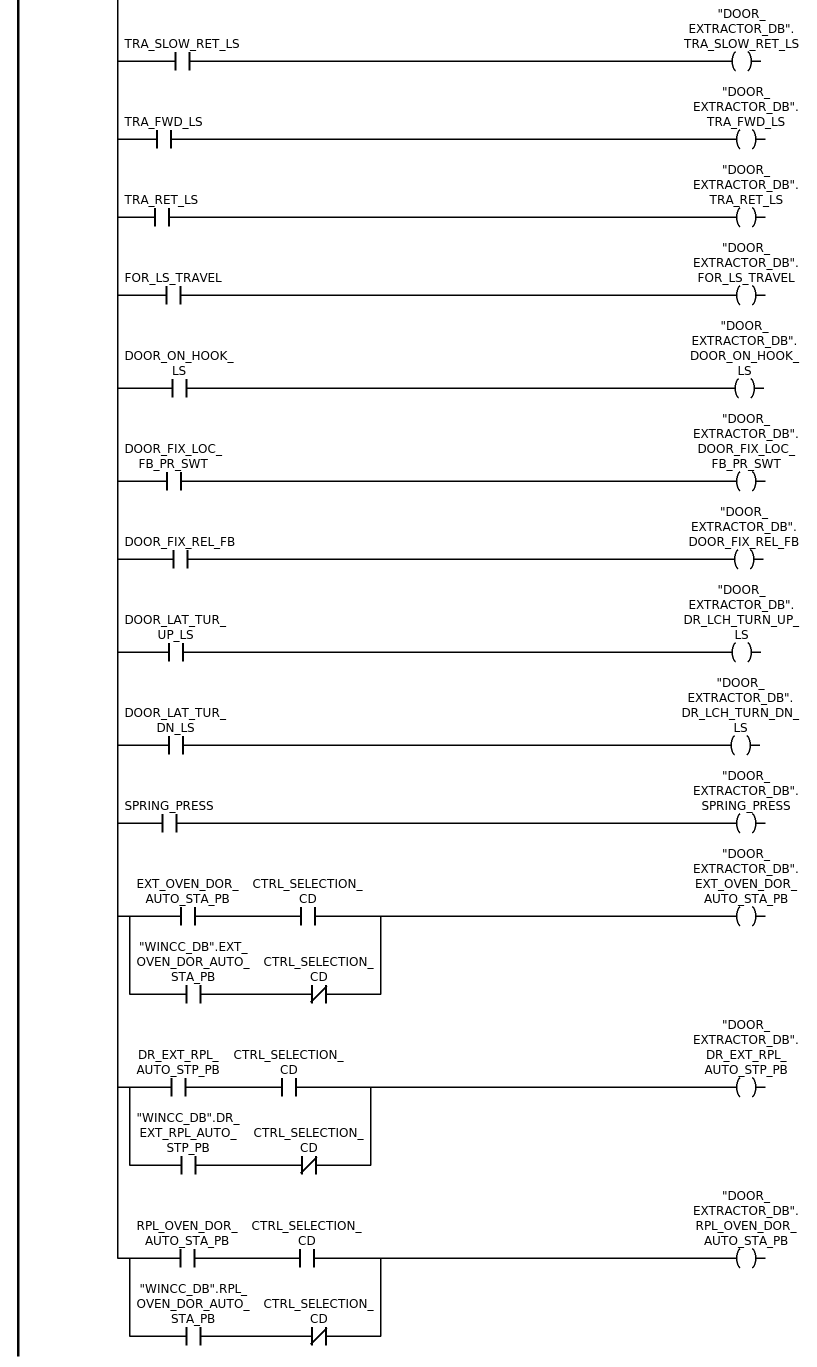
[picture p24: INPUT_MAPPING networks 13-13]
NETWORK
TITLE =
      A     "ALWAYS_ON";
      =     L 0.0;
      A     L 0.0;
      A(;
      O     "DOOR_EXT_LOC_SS";
      O;
      A     "WINCC_DB".REPAIR_MODE_SS;
      AN    "CTRL_SELECTION_CD";
      );
      =     "DOOR_EXTRACTOR_DB".DOOR_EXT_LOC_SS;
      A     L 0.0;
      A(;
      A     "DOOR_EXT_MAN_SS";
      A     "CTRL_SELECTION_CD";
      O;
      A     "WINCC_DB".DE_MAN_SS;
      AN    "DOOR_EXTRACTOR_DB".DOOR_EXT_LOC_SS;
      A     "WINCC_DB".OPER_MODE_SS;
      AN    "CTRL_SELECTION_CD";
      );
      =     "DOOR_EXTRACTOR_DB".DOOR_EXT_MAN_SS;
      A     L 0.0;
      A(;
      A     "DOOR_EXT_AUTO_SS";
      A     "CTRL_SELECTION_CD";
      O;
      A     "WINCC_DB".DE_AUTO_SS;
      AN    "DOOR_EXTRACTOR_DB".DOOR_EXT_LOC_SS;
      A     "WINCC_DB".OPER_MODE_SS;
      AN    "CTRL_SELECTION_CD";
      );
      =     "DOOR_EXTRACTOR_DB".DOOR_EXT_AUTO_SS;
      A     L 0.0;
      A     "WINCC_DB".DE_AUTO_MAN_SS_TAG;
      =     "WINCC_DB".DE_AUTO_SS;
      A     L 0.0;
      AN    "WINCC_DB".DE_AUTO_MAN_SS_TAG;
      =     "WINCC_DB".DE_MAN_SS;
      A     L 0.0;
      A(;
      A     "DOOR_EXT_STP_PB";
      A     "CTRL_SELECTION_CD";
      O;
      A     "WINCC_DB".DE_STP_PB;
      AN    "CTRL_SELECTION_CD";
      );
      =     "DOOR_EXTRACTOR_DB".DOOR_EXT_STP_PB;
      A     L 0.0;
      A(;
      A     "SLEW_FWD_STA_PB";
      A     "CTRL_SELECTION_CD";
      O;
      A     "WINCC_DB".SLEW_FWD_STA_PB;
      AN    "CTRL_SELECTION_CD";
      );
      =     "DOOR_EXTRACTOR_DB".SLEW_FWD_STA_PB;
      A     L 0.0;
      A(;
      A     "SLEW_RET_STA_PB";
      A     "CTRL_SELECTION_CD";
      O;
      A     "WINCC_DB".SLEW_RET_STA_PB;
      AN    "CTRL_SELECTION_CD";
      );
      =     "DOOR_EXTRACTOR_DB".SLEW_RET_STA_PB;
      A     L 0.0;
      A(;
      A     "VER_COMP_FWD_STA";
      A     "CTRL_SELECTION_CD";
      O;
      A     "WINCC_DB".VER_COMP_FWD_STA_PB;
      AN    "CTRL_SELECTION_CD";
      );
      =     "DOOR_EXTRACTOR_DB".VER_COMP_FWD_STA_PB;
      A     L 0.0;
      A(;
      A     "VER_COMP_RET_STA";
      A     "CTRL_SELECTION_CD";
      O;
      A     "WINCC_DB".VER_COMP_RET_STA_PB;
      AN    "CTRL_SELECTION_CD";
      );
      =     "DOOR_EXTRACTOR_DB".VER_COMP_RET_STA_PB;
      A     L 0.0;
      A(;
      A     "TRA_FWD_STA";
      A     "CTRL_SELECTION_CD";
      O;
      A     "WINCC_DB".TRA_FWD_STA_PB;
      AN    "CTRL_SELECTION_CD";
      );
      =     "DOOR_EXTRACTOR_DB".TRA_FWD_STA_PB;
      A     L 0.0;
      A(;
      A     "TRA_RET_STA";
      A     "CTRL_SELECTION_CD";
      O;
      A     "WINCC_DB".TRA_RET_STA_PB;
      AN    "CTRL_SELECTION_CD";
      );
      =     "DOOR_EXTRACTOR_DB".TRA_RET_STA_PB;
      A     L 0.0;
      A(;
      A     "MAN_STK_UP_STA_PB";
      A     "CTRL_SELECTION_CD";
      O;
      A     "WINCC_DB".MAIN_STK_UP_STA_PB;
      AN    "CTRL_SELECTION_CD";
      );
      =     "DOOR_EXTRACTOR_DB".MAIN_STK_UP_STA_PB;
      A     L 0.0;
      A(;
      A     "MAN_STK_UP_DN_PB";
      A     "CTRL_SELECTION_CD";
      O;
      A     "WINCC_DB".MAIN_STK_UP_DN_PB;
      AN    "CTRL_SELECTION_CD";
      );
      =     "DOOR_EXTRACTOR_DB".MAIN_STK_UP_DN_PB;
      A     L 0.0;
      A(;
      A     "FNL_STK_UP_STA_PB";
      A     "CTRL_SELECTION_CD";
      O;
      A     "WINCC_DB".FIN_STK_UP_STA_PB;
      AN    "CTRL_SELECTION_CD";
      );
      =     "DOOR_EXTRACTOR_DB".FIN_STK_UP_STA_PB;
      A     L 0.0;
      A(;
      A     "FNL_STK_UP_DN_PB";
      A     "CTRL_SELECTION_CD";
      O;
      A     "WINCC_DB".FIN_STK_UP_DN_PB;
      AN    "CTRL_SELECTION_CD";
      );
      =     "DOOR_EXTRACTOR_DB".FIN_STK_UP_DN_PB;
      A     L 0.0;
      A(;
      A     "PRE_STK_UP_STA_PB";
      A     "CTRL_SELECTION_CD";
      O;
      A     "WINCC_DB".PRE_STK_UP_STA_PB;
      AN    "CTRL_SELECTION_CD";
      );
      =     "DOOR_EXTRACTOR_DB".PRE_STK_UP_STA_PB;
      A     L 0.0;
      A(;
      A     "PRE_STK_UP_DN_PB";
      A     "CTRL_SELECTION_CD";
      O;
      A     "WINCC_DB".PRE_STK_UP_DN_PB;
      AN    "CTRL_SELECTION_CD";
      );
      =     "DOOR_EXTRACTOR_DB".PRE_STK_UP_DN_PB;
      A     L 0.0;
      A(;
      A     "DOOR_SPRG_PRS_STA_PB";
      A     "CTRL_SELECTION_CD";
      O;
      A     "WINCC_DB".DR_SPNG_LK_STA_PB;
      AN    "CTRL_SELECTION_CD";
      );
      =     "DOOR_EXTRACTOR_DB".DR_SPNG_LK_STA_PB;
      A     L 0.0;
      A(;
      A     "DOOR_SPRG_RLES_STA_PB";
      A     "CTRL_SELECTION_CD";
      O;
      A     "WINCC_DB".DR_SPNG_UNLK_STA_PB;
      AN    "CTRL_SELECTION_CD";
      );
      =     "DOOR_EXTRACTOR_DB".DR_SPNG_UNLK_STA_PB;
      A     L 0.0;
      A(;
      A     "DOOR_LCH_TURN_LOCK";
      A     "CTRL_SELECTION_CD";
      O;
      A     "WINCC_DB".DR_LCH_TURN_UP_PB;
      AN    "CTRL_SELECTION_CD";
      );
      =     "DOOR_EXTRACTOR_DB".DR_LCH_TURN_UP_PB;
      A     L 0.0;
      A(;
      A     "DOOR_LCH_TURN_UNLOC";
      A     "CTRL_SELECTION_CD";
      O;
      A     "WINCC_DB".DR_LCH_TURN_DN_PB;
      AN    "CTRL_SELECTION_CD";
      );
      =     "DOOR_EXTRACTOR_DB".DR_LCH_TURN_DN_PB;
      A     L 0.0;
      A     "EMERGENCY_PB_LCS_73";
      =     "DOOR_EXTRACTOR_DB".EMERGENCY_PB_LCS_73;
      A     L 0.0;
      A     "SLEW_FWD_STA_LCS";
      =     "DOOR_EXTRACTOR_DB".SLEW_FWD_STA_PB_LCS;
      A     L 0.0;
      A     "SLEW_RET_STA_LCS";
      =     "DOOR_EXTRACTOR_DB".SLEW_RET_STA_PB_LCS;
      A     L 0.0;
      A     "VER_COMP_FWD_STA_LCS";
      =     "DOOR_EXTRACTOR_DB".VER_COMP_FWD_STA_PB_LCS;
      A     L 0.0;
      A     "VER_COMP_RET_STA_LCS";
      =     "DOOR_EXTRACTOR_DB".VER_COMP_RET_STA_PB_LCS;
      A     L 0.0;
      A     "TRA_FWD_STA_LCS";
      =     "DOOR_EXTRACTOR_DB".TRA_FWD_STA_PB_LCS;
      A     L 0.0;
      A     "TRA_BACK_STA_LCS";
      =     "DOOR_EXTRACTOR_DB".TRA_RET_STA_PB_LCS;
      A     L 0.0;
      A     "MAIN_STK_UP_STA_LCS";
      =     "DOOR_EXTRACTOR_DB".MAIN_STK_UP_STA_PB_LCS;
      A     L 0.0;
      A     "MAIN_STK_DN_STA_LCS";
      =     "DOOR_EXTRACTOR_DB".MAIN_STK_DN_STA_PB_LCS;
      A     L 0.0;
      A     "FNL_STK_UP_STA_LCS";
      =     "DOOR_EXTRACTOR_DB".FIN_STK_UP_STA_PB_LCS;
      A     L 0.0;
      A     "FNL_STK_DN_STA_LCS";
      =     "DOOR_EXTRACTOR_DB".FIN_STK_DN_STA_PB_LCS;
      A     L 0.0;
      A     "PRE_STK_UP_STA_LCS";
      =     "DOOR_EXTRACTOR_DB".PRE_STK_UP_STA_PB_LCS;
      A     L 0.0;
      A     "PRE_STK_DN_STA_LCS";
      =     "DOOR_EXTRACTOR_DB".PRE_STK_DN_STA_PB_LCS;
      A     L 0.0;
      A     "DOOR_SPRG_PRS_LK_STA_LCS";
      =     "DOOR_EXTRACTOR_DB".DR_SPNG_LK_STA_PB_LCS;
      A     L 0.0;
      A     "DOOR_SPRG_RLES_UNLSTA_LC";
      =     "DOOR_EXTRACTOR_DB".DR_SPNG_UNLK_STA_PB_LCS;
      A     L 0.0;
      A     "LAMP_TEST_PB_LCS_73";
      =     "DOOR_EXTRACTOR_DB".LAMP_TEST_PB_LCS_73;
      A     L 0.0;
      A     "DOOR_LAT_LOCK_PB_LCS";
      =     "DOOR_EXTRACTOR_DB".DR_LCH_TURN_UP_PB_LCS;
      A     L 0.0;
      A     "DOOR_LAT_UNLOCK_PB_LCS1";
      =     "DOOR_EXTRACTOR_DB".DR_LCH_TURN_DN_PB_LCS;
      A     L 0.0;
      A     "DOOR_LAT_HOME_PB_LCS";
      =     "DOOR_EXTRACTOR_DB".DR_LCH_TURN_HOME_PB_LCS;
      A     L 0.0;
      A     "SLEW_SLOW_FWD_LS";
      =     "DOOR_EXTRACTOR_DB".SLEW_SLOW_FWD_LS;
      A     L 0.0;
      A     "SLEW_SLOW_RET_LS";
      =     "DOOR_EXTRACTOR_DB".SLEW_SLOW_RET_LS;
      A     L 0.0;
      A     "SLEW_NOR_FWD_LS";
      =     "DOOR_EXTRACTOR_DB".SLEW_NOR_FWD_LS;
      A     L 0.0;
      A     "SLEW_NOR_RET_LS";
      =     "DOOR_EXTRACTOR_DB".SLEW_NOR_RET_LS;
      A     L 0.0;
      A     "TRA_SLOW_FWD_LS";
      =     "DOOR_EXTRACTOR_DB".TRA_SLOW_FWD_LS;
      A     L 0.0;
      A     "TRA_SLOW_RET_LS";
      =     "DOOR_EXTRACTOR_DB".TRA_SLOW_RET_LS;
      A     L 0.0;
      A     "TRA_FWD_LS";
      =     "DOOR_EXTRACTOR_DB".TRA_FWD_LS;
      A     L 0.0;
      A     "TRA_RET_LS";
      =     "DOOR_EXTRACTOR_DB".TRA_RET_LS;
      A     L 0.0;
      A     "FOR_LS_TRAVEL";
      =     "DOOR_EXTRACTOR_DB".FOR_LS_TRAVEL;
      A     L 0.0;
      A     "DOOR_ON_HOOK_LS";
      =     "DOOR_EXTRACTOR_DB".DOOR_ON_HOOK_LS;
      A     L 0.0;
      A     "DOOR_FIX_LOC_FB_PR_SWT";
      =     "DOOR_EXTRACTOR_DB".DOOR_FIX_LOC_FB_PR_SWT;
      A     L 0.0;
      A     "DOOR_FIX_REL_FB";
      =     "DOOR_EXTRACTOR_DB".DOOR_FIX_REL_FB;
      A     L 0.0;
      A     "DOOR_LAT_TUR_UP_LS";
      =     "DOOR_EXTRACTOR_DB".DR_LCH_TURN_UP_LS;
      A     L 0.0;
      A     "DOOR_LAT_TUR_DN_LS";
      =     "DOOR_EXTRACTOR_DB".DR_LCH_TURN_DN_LS;
      A     L 0.0;
      A     "SPRING_PRESS";
      =     "DOOR_EXTRACTOR_DB".SPRING_PRESS;
      A     L 0.0;
      A(;
      A     "EXT_OVEN_DOR_AUTO_STA_PB";
      A     "CTRL_SELECTION_CD";
      O;
      A     "WINCC_DB".EXT_OVEN_DOR_AUTO_STA_PB;
      AN    "CTRL_SELECTION_CD";
      );
      =     "DOOR_EXTRACTOR_DB".EXT_OVEN_DOR_AUTO_STA_PB;
      A     L 0.0;
      A(;
      A     "DR_EXT_RPL_AUTO_STP_PB";
      A     "CTRL_SELECTION_CD";
      O;
      A     "WINCC_DB".DR_EXT_RPL_AUTO_STP_PB;
      AN    "CTRL_SELECTION_CD";
      );
      =     "DOOR_EXTRACTOR_DB".DR_EXT_RPL_AUTO_STP_PB;
      A     L 0.0;
      A(;
      A     "RPL_OVEN_DOR_AUTO_STA_PB";
      A     "CTRL_SELECTION_CD";
      O;
      A     "WINCC_DB".RPL_OVEN_DOR_AUTO_STA_PB;
      AN    "CTRL_SELECTION_CD";
      );
      =     "DOOR_EXTRACTOR_DB".RPL_OVEN_DOR_AUTO_STA_PB;
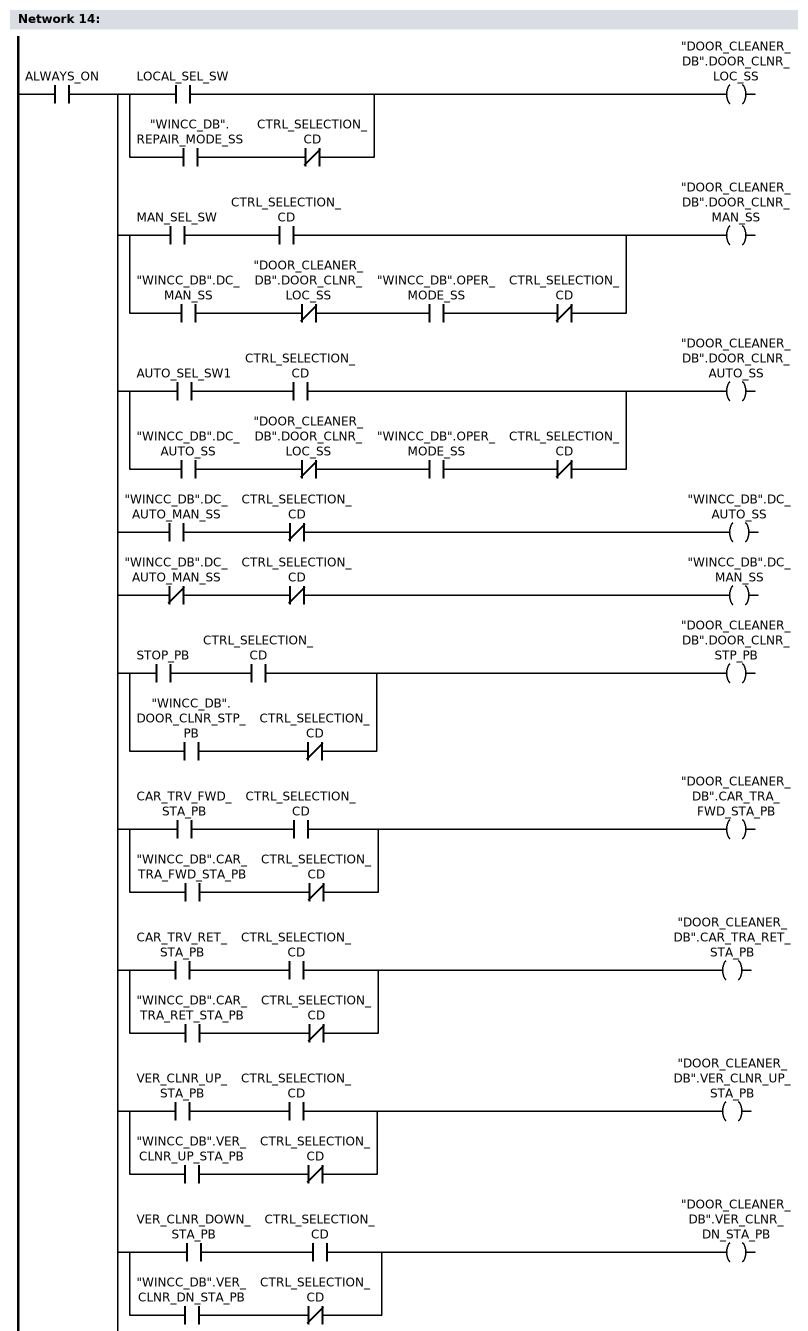
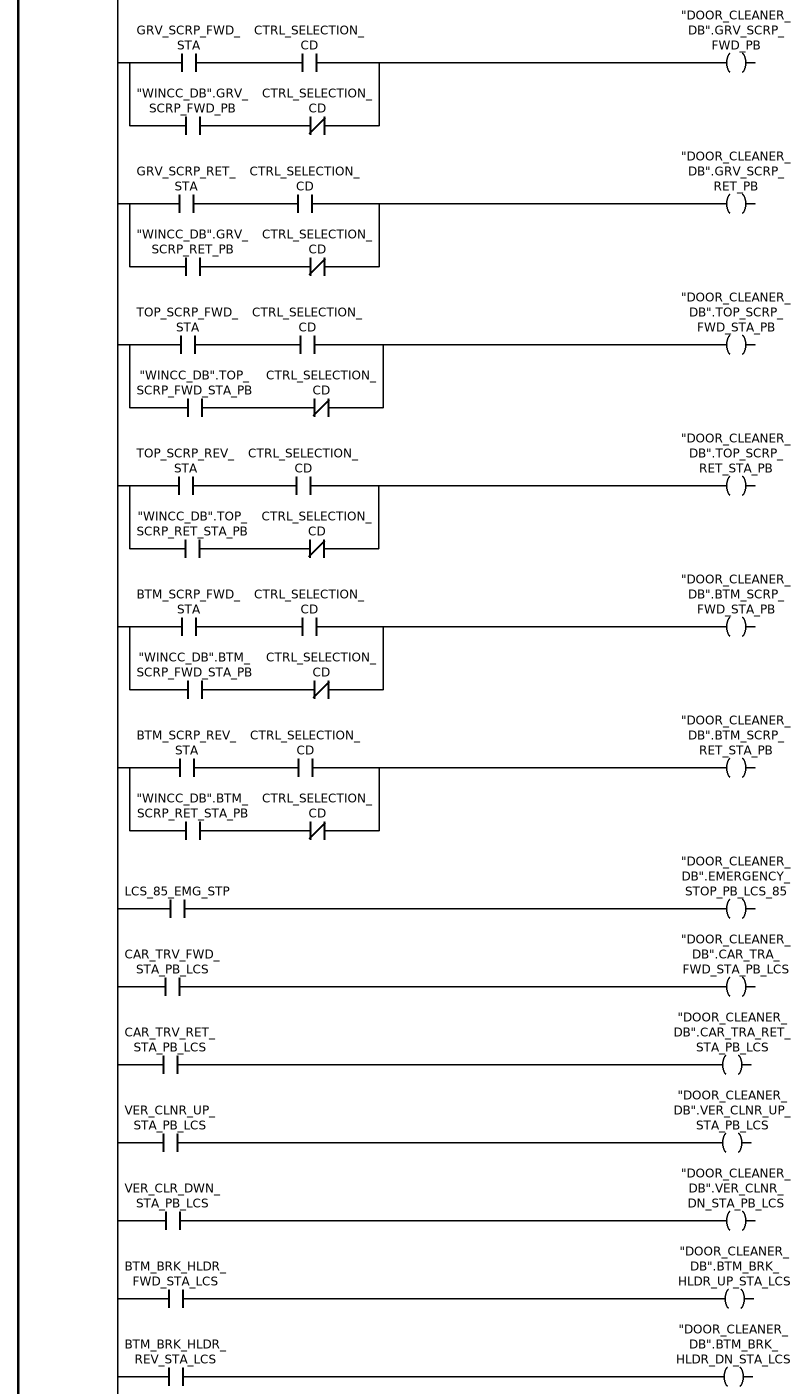
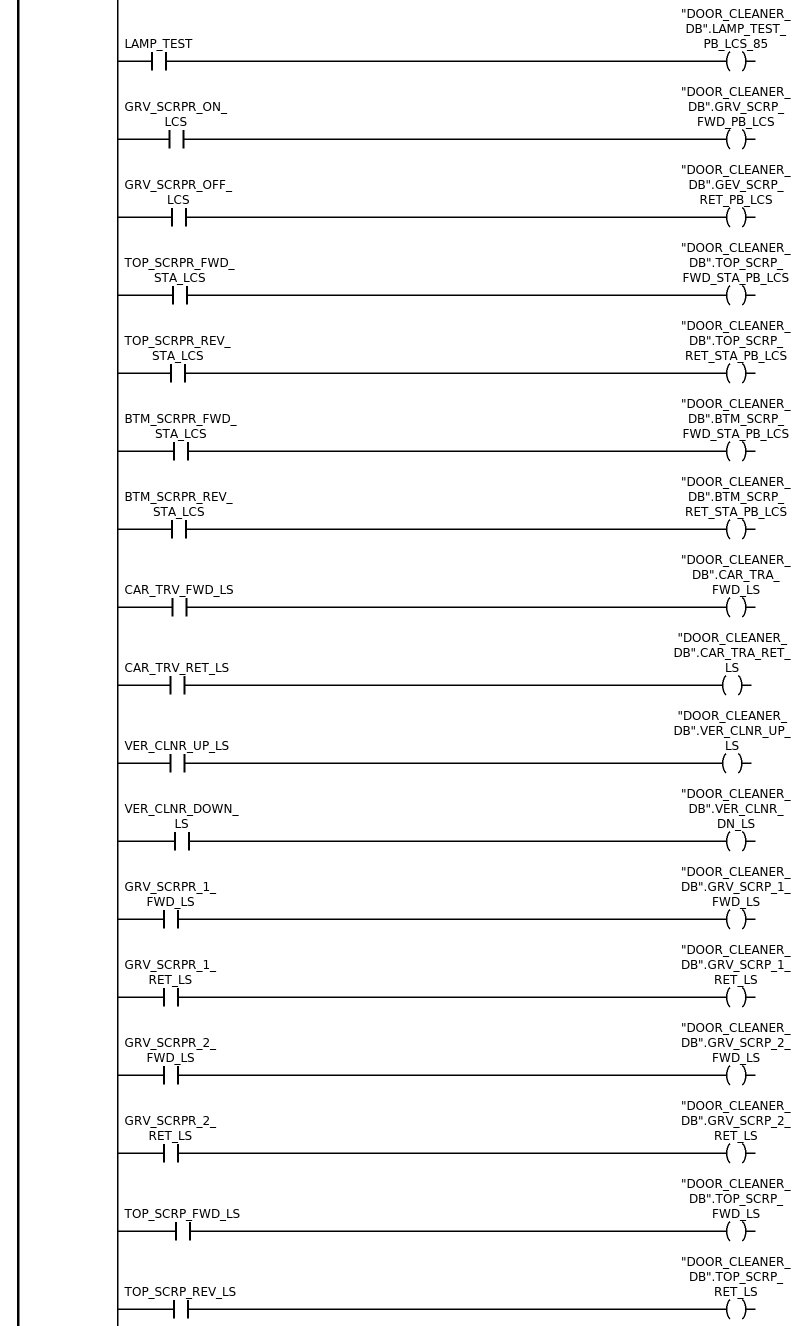
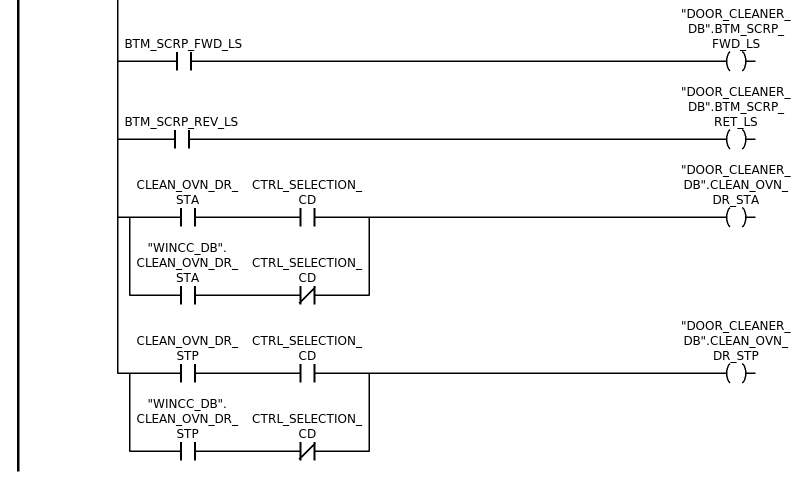
NETWORK
TITLE =
      A     "ALWAYS_ON";
      =     L 0.0;
      A     L 0.0;
      A(;
      O     "LOCAL_SEL_SW";
      O;
      A     "WINCC_DB".REPAIR_MODE_SS;
      AN    "CTRL_SELECTION_CD";
      );
      =     "DOOR_CLEANER_DB".DOOR_CLNR_LOC_SS;
      A     L 0.0;
      A(;
      A     "MAN_SEL_SW";
      A     "CTRL_SELECTION_CD";
      O;
      A     "WINCC_DB".DC_MAN_SS;
      AN    "DOOR_CLEANER_DB".DOOR_CLNR_LOC_SS;
      A     "WINCC_DB".OPER_MODE_SS;
      AN    "CTRL_SELECTION_CD";
      );
      =     "DOOR_CLEANER_DB".DOOR_CLNR_MAN_SS;
      A     L 0.0;
      A(;
      A     "AUTO_SEL_SW1";
      A     "CTRL_SELECTION_CD";
      O;
      A     "WINCC_DB".DC_AUTO_SS;
      AN    "DOOR_CLEANER_DB".DOOR_CLNR_LOC_SS;
      A     "WINCC_DB".OPER_MODE_SS;
      AN    "CTRL_SELECTION_CD";
      );
      =     "DOOR_CLEANER_DB".DOOR_CLNR_AUTO_SS;
      A     L 0.0;
      A     "WINCC_DB".DC_AUTO_MAN_SS;
      AN    "CTRL_SELECTION_CD";
      =     "WINCC_DB".DC_AUTO_SS;
      A     L 0.0;
      AN    "WINCC_DB".DC_AUTO_MAN_SS;
      AN    "CTRL_SELECTION_CD";
      =     "WINCC_DB".DC_MAN_SS;
      A     L 0.0;
      A(;
      A     "STOP_PB";
      A     "CTRL_SELECTION_CD";
      O;
      A     "WINCC_DB".DOOR_CLNR_STP_PB;
      AN    "CTRL_SELECTION_CD";
      );
      =     "DOOR_CLEANER_DB".DOOR_CLNR_STP_PB;
      A     L 0.0;
      A(;
      A     "CAR_TRV_FWD_STA_PB";
      A     "CTRL_SELECTION_CD";
      O;
      A     "WINCC_DB".CAR_TRA_FWD_STA_PB;
      AN    "CTRL_SELECTION_CD";
      );
      =     "DOOR_CLEANER_DB".CAR_TRA_FWD_STA_PB;
      A     L 0.0;
      A(;
      A     "CAR_TRV_RET_STA_PB";
      A     "CTRL_SELECTION_CD";
      O;
      A     "WINCC_DB".CAR_TRA_RET_STA_PB;
      AN    "CTRL_SELECTION_CD";
      );
      =     "DOOR_CLEANER_DB".CAR_TRA_RET_STA_PB;
      A     L 0.0;
      A(;
      A     "VER_CLNR_UP_STA_PB";
      A     "CTRL_SELECTION_CD";
      O;
      A     "WINCC_DB".VER_CLNR_UP_STA_PB;
      AN    "CTRL_SELECTION_CD";
      );
      =     "DOOR_CLEANER_DB".VER_CLNR_UP_STA_PB;
      A     L 0.0;
      A(;
      A     "VER_CLNR_DOWN_STA_PB";
      A     "CTRL_SELECTION_CD";
      O;
      A     "WINCC_DB".VER_CLNR_DN_STA_PB;
      AN    "CTRL_SELECTION_CD";
      );
      =     "DOOR_CLEANER_DB".VER_CLNR_DN_STA_PB;
      A     L 0.0;
      A(;
      A     "GRV_SCRP_FWD_STA";
      A     "CTRL_SELECTION_CD";
      O;
      A     "WINCC_DB".GRV_SCRP_FWD_PB;
      AN    "CTRL_SELECTION_CD";
      );
      =     "DOOR_CLEANER_DB".GRV_SCRP_FWD_PB;
      A     L 0.0;
      A(;
      A     "GRV_SCRP_RET_STA";
      A     "CTRL_SELECTION_CD";
      O;
      A     "WINCC_DB".GRV_SCRP_RET_PB;
      AN    "CTRL_SELECTION_CD";
      );
      =     "DOOR_CLEANER_DB".GRV_SCRP_RET_PB;
      A     L 0.0;
      A(;
      A     "TOP_SCRP_FWD_STA";
      A     "CTRL_SELECTION_CD";
      O;
      A     "WINCC_DB".TOP_SCRP_FWD_STA_PB;
      AN    "CTRL_SELECTION_CD";
      );
      =     "DOOR_CLEANER_DB".TOP_SCRP_FWD_STA_PB;
      A     L 0.0;
      A(;
      A     "TOP_SCRP_REV_STA";
      A     "CTRL_SELECTION_CD";
      O;
      A     "WINCC_DB".TOP_SCRP_RET_STA_PB;
      AN    "CTRL_SELECTION_CD";
      );
      =     "DOOR_CLEANER_DB".TOP_SCRP_RET_STA_PB;
      A     L 0.0;
      A(;
      A     "BTM_SCRP_FWD_STA";
      A     "CTRL_SELECTION_CD";
      O;
      A     "WINCC_DB".BTM_SCRP_FWD_STA_PB;
      AN    "CTRL_SELECTION_CD";
      );
      =     "DOOR_CLEANER_DB".BTM_SCRP_FWD_STA_PB;
      A     L 0.0;
      A(;
      A     "BTM_SCRP_REV_STA";
      A     "CTRL_SELECTION_CD";
      O;
      A     "WINCC_DB".BTM_SCRP_RET_STA_PB;
      AN    "CTRL_SELECTION_CD";
      );
      =     "DOOR_CLEANER_DB".BTM_SCRP_RET_STA_PB;
      A     L 0.0;
      A     "LCS_85_EMG_STP";
      =     "DOOR_CLEANER_DB".EMERGENCY_STOP_PB_LCS_85;
      A     L 0.0;
      A     "CAR_TRV_FWD_STA_PB_LCS";
      =     "DOOR_CLEANER_DB".CAR_TRA_FWD_STA_PB_LCS;
      A     L 0.0;
      A     "CAR_TRV_RET_STA_PB_LCS";
      =     "DOOR_CLEANER_DB".CAR_TRA_RET_STA_PB_LCS;
      A     L 0.0;
      A     "VER_CLNR_UP_STA_PB_LCS";
      =     "DOOR_CLEANER_DB".VER_CLNR_UP_STA_PB_LCS;
      A     L 0.0;
      A     "VER_CLR_DWN_STA_PB_LCS";
      =     "DOOR_CLEANER_DB".VER_CLNR_DN_STA_PB_LCS;
      A     L 0.0;
      A     "BTM_BRK_HLDR_FWD_STA_LCS";
      =     "DOOR_CLEANER_DB".BTM_BRK_HLDR_UP_STA_LCS;
      A     L 0.0;
      A     "BTM_BRK_HLDR_REV_STA_LCS";
      =     "DOOR_CLEANER_DB".BTM_BRK_HLDR_DN_STA_LCS;
      A     L 0.0;
      A     "LAMP_TEST";
      =     "DOOR_CLEANER_DB".LAMP_TEST_PB_LCS_85;
      A     L 0.0;
      A     "GRV_SCRPR_ON_LCS";
      =     "DOOR_CLEANER_DB".GRV_SCRP_FWD_PB_LCS;
      A     L 0.0;
      A     "GRV_SCRPR_OFF_LCS";
      =     "DOOR_CLEANER_DB".GEV_SCRP_RET_PB_LCS;
      A     L 0.0;
      A     "TOP_SCRPR_FWD_STA_LCS";
      =     "DOOR_CLEANER_DB".TOP_SCRP_FWD_STA_PB_LCS;
      A     L 0.0;
      A     "TOP_SCRPR_REV_STA_LCS";
      =     "DOOR_CLEANER_DB".TOP_SCRP_RET_STA_PB_LCS;
      A     L 0.0;
      A     "BTM_SCRPR_FWD_STA_LCS";
      =     "DOOR_CLEANER_DB".BTM_SCRP_FWD_STA_PB_LCS;
      A     L 0.0;
      A     "BTM_SCRPR_REV_STA_LCS";
      =     "DOOR_CLEANER_DB".BTM_SCRP_RET_STA_PB_LCS;
      A     L 0.0;
      A     "CAR_TRV_FWD_LS";
      =     "DOOR_CLEANER_DB".CAR_TRA_FWD_LS;
      A     L 0.0;
      A     "CAR_TRV_RET_LS";
      =     "DOOR_CLEANER_DB".CAR_TRA_RET_LS;
      A     L 0.0;
      A     "VER_CLNR_UP_LS";
      =     "DOOR_CLEANER_DB".VER_CLNR_UP_LS;
      A     L 0.0;
      A     "VER_CLNR_DOWN_LS";
      =     "DOOR_CLEANER_DB".VER_CLNR_DN_LS;
      A     L 0.0;
      A     "GRV_SCRPR_1_FWD_LS";
      =     "DOOR_CLEANER_DB".GRV_SCRP_1_FWD_LS;
      A     L 0.0;
      A     "GRV_SCRPR_1_RET_LS";
      =     "DOOR_CLEANER_DB".GRV_SCRP_1_RET_LS;
      A     L 0.0;
      A     "GRV_SCRPR_2_FWD_LS";
      =     "DOOR_CLEANER_DB".GRV_SCRP_2_FWD_LS;
      A     L 0.0;
      A     "GRV_SCRPR_2_RET_LS";
      =     "DOOR_CLEANER_DB".GRV_SCRP_2_RET_LS;
      A     L 0.0;
      A     "TOP_SCRP_FWD_LS";
      =     "DOOR_CLEANER_DB".TOP_SCRP_FWD_LS;
      A     L 0.0;
      A     "TOP_SCRP_REV_LS";
      =     "DOOR_CLEANER_DB".TOP_SCRP_RET_LS;
      A     L 0.0;
      A     "BTM_SCRP_FWD_LS";
      =     "DOOR_CLEANER_DB".BTM_SCRP_FWD_LS;
      A     L 0.0;
      A     "BTM_SCRP_REV_LS";
      =     "DOOR_CLEANER_DB".BTM_SCRP_RET_LS;
      A     L 0.0;
      A(;
      A     "CLEAN_OVN_DR_STA";
      A     "CTRL_SELECTION_CD";
      O;
      A     "WINCC_DB".CLEAN_OVN_DR_STA;
      AN    "CTRL_SELECTION_CD";
      );
      =     "DOOR_CLEANER_DB".CLEAN_OVN_DR_STA;
      A     L 0.0;
      A(;
      A     "CLEAN_OVN_DR_STP";
      A     "CTRL_SELECTION_CD";
      O;
      A     "WINCC_DB".CLEAN_OVN_DR_STP;
      AN    "CTRL_SELECTION_CD";
      );
      =     "DOOR_CLEANER_DB".CLEAN_OVN_DR_STP;
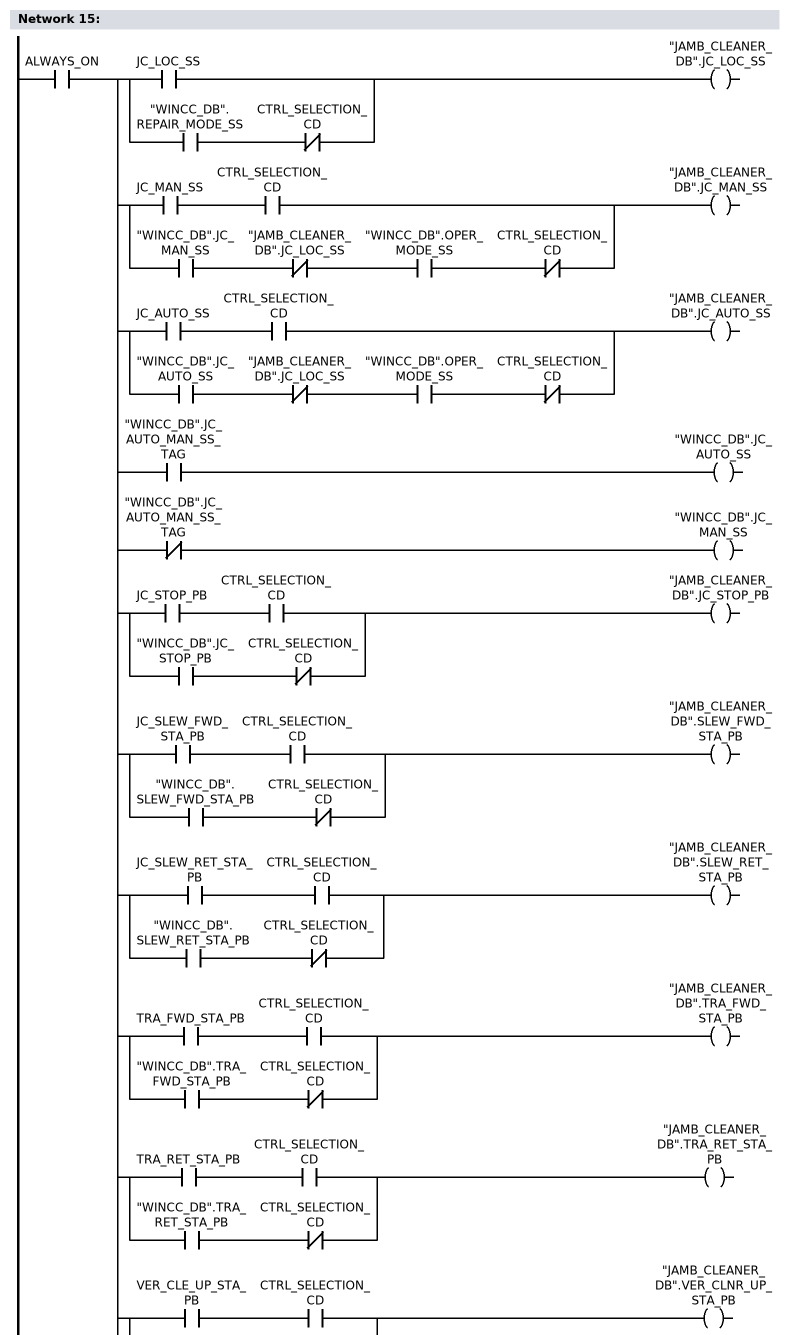
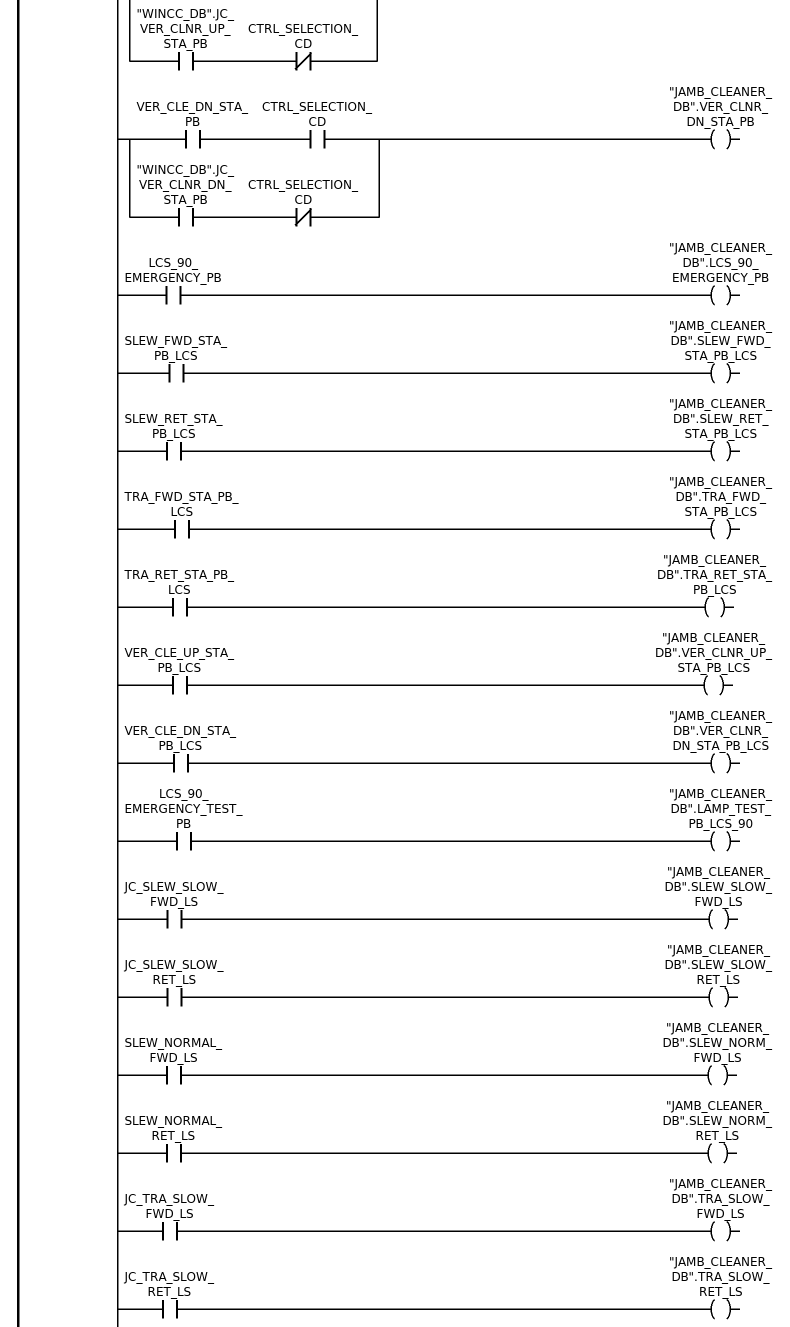
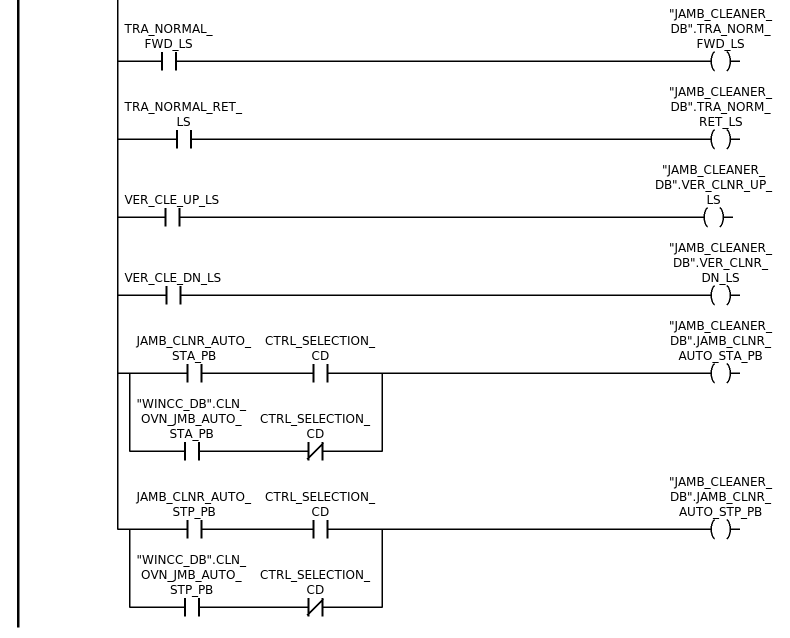
NETWORK
TITLE =
      A     "ALWAYS_ON";
      =     L 0.0;
      A     L 0.0;
      A(;
      O     "JC_LOC_SS";
      O;
      A     "WINCC_DB".REPAIR_MODE_SS;
      AN    "CTRL_SELECTION_CD";
      );
      =     "JAMB_CLEANER_DB".JC_LOC_SS;
      A     L 0.0;
      A(;
      A     "JC_MAN_SS";
      A     "CTRL_SELECTION_CD";
      O;
      A     "WINCC_DB".JC_MAN_SS;
      AN    "JAMB_CLEANER_DB".JC_LOC_SS;
      A     "WINCC_DB".OPER_MODE_SS;
      AN    "CTRL_SELECTION_CD";
      );
      =     "JAMB_CLEANER_DB".JC_MAN_SS;
      A     L 0.0;
      A(;
      A     "JC_AUTO_SS";
      A     "CTRL_SELECTION_CD";
      O;
      A     "WINCC_DB".JC_AUTO_SS;
      AN    "JAMB_CLEANER_DB".JC_LOC_SS;
      A     "WINCC_DB".OPER_MODE_SS;
      AN    "CTRL_SELECTION_CD";
      );
      =     "JAMB_CLEANER_DB".JC_AUTO_SS;
      A     L 0.0;
      A     "WINCC_DB".JC_AUTO_MAN_SS_TAG;
      =     "WINCC_DB".JC_AUTO_SS;
      A     L 0.0;
      AN    "WINCC_DB".JC_AUTO_MAN_SS_TAG;
      =     "WINCC_DB".JC_MAN_SS;
      A     L 0.0;
      A(;
      A     "JC_STOP_PB";
      A     "CTRL_SELECTION_CD";
      O;
      A     "WINCC_DB".JC_STOP_PB;
      AN    "CTRL_SELECTION_CD";
      );
      =     "JAMB_CLEANER_DB".JC_STOP_PB;
      A     L 0.0;
      A(;
      A     "JC_SLEW_FWD_STA_PB";
      A     "CTRL_SELECTION_CD";
      O;
      A     "WINCC_DB".SLEW_FWD_STA_PB;
      AN    "CTRL_SELECTION_CD";
      );
      =     "JAMB_CLEANER_DB".SLEW_FWD_STA_PB;
      A     L 0.0;
      A(;
      A     "JC_SLEW_RET_STA_PB";
      A     "CTRL_SELECTION_CD";
      O;
      A     "WINCC_DB".SLEW_RET_STA_PB;
      AN    "CTRL_SELECTION_CD";
      );
      =     "JAMB_CLEANER_DB".SLEW_RET_STA_PB;
      A     L 0.0;
      A(;
      A     "TRA_FWD_STA_PB";
      A     "CTRL_SELECTION_CD";
      O;
      A     "WINCC_DB".TRA_FWD_STA_PB;
      AN    "CTRL_SELECTION_CD";
      );
      =     "JAMB_CLEANER_DB".TRA_FWD_STA_PB;
      A     L 0.0;
      A(;
      A     "TRA_RET_STA_PB";
      A     "CTRL_SELECTION_CD";
      O;
      A     "WINCC_DB".TRA_RET_STA_PB;
      AN    "CTRL_SELECTION_CD";
      );
      =     "JAMB_CLEANER_DB".TRA_RET_STA_PB;
      A     L 0.0;
      A(;
      A     "VER_CLE_UP_STA_PB";
      A     "CTRL_SELECTION_CD";
      O;
      A     "WINCC_DB".JC_VER_CLNR_UP_STA_PB;
      AN    "CTRL_SELECTION_CD";
      );
      =     "JAMB_CLEANER_DB".VER_CLNR_UP_STA_PB;
      A     L 0.0;
      A(;
      A     "VER_CLE_DN_STA_PB";
      A     "CTRL_SELECTION_CD";
      O;
      A     "WINCC_DB".JC_VER_CLNR_DN_STA_PB;
      AN    "CTRL_SELECTION_CD";
      );
      =     "JAMB_CLEANER_DB".VER_CLNR_DN_STA_PB;
      A     L 0.0;
      A     "LCS_90_EMERGENCY_PB";
      =     "JAMB_CLEANER_DB".LCS_90_EMERGENCY_PB;
      A     L 0.0;
      A     "SLEW_FWD_STA_PB_LCS";
      =     "JAMB_CLEANER_DB".SLEW_FWD_STA_PB_LCS;
      A     L 0.0;
      A     "SLEW_RET_STA_PB_LCS";
      =     "JAMB_CLEANER_DB".SLEW_RET_STA_PB_LCS;
      A     L 0.0;
      A     "TRA_FWD_STA_PB_LCS";
      =     "JAMB_CLEANER_DB".TRA_FWD_STA_PB_LCS;
      A     L 0.0;
      A     "TRA_RET_STA_PB_LCS";
      =     "JAMB_CLEANER_DB".TRA_RET_STA_PB_LCS;
      A     L 0.0;
      A     "VER_CLE_UP_STA_PB_LCS";
      =     "JAMB_CLEANER_DB".VER_CLNR_UP_STA_PB_LCS;
      A     L 0.0;
      A     "VER_CLE_DN_STA_PB_LCS";
      =     "JAMB_CLEANER_DB".VER_CLNR_DN_STA_PB_LCS;
      A     L 0.0;
      A     "LCS_90_EMERGENCY_TEST_PB";
      =     "JAMB_CLEANER_DB".LAMP_TEST_PB_LCS_90;
      A     L 0.0;
      A     "JC_SLEW_SLOW_FWD_LS";
      =     "JAMB_CLEANER_DB".SLEW_SLOW_FWD_LS;
      A     L 0.0;
      A     "JC_SLEW_SLOW_RET_LS";
      =     "JAMB_CLEANER_DB".SLEW_SLOW_RET_LS;
      A     L 0.0;
      A     "SLEW_NORMAL_FWD_LS";
      =     "JAMB_CLEANER_DB".SLEW_NORM_FWD_LS;
      A     L 0.0;
      A     "SLEW_NORMAL_RET_LS";
      =     "JAMB_CLEANER_DB".SLEW_NORM_RET_LS;
      A     L 0.0;
      A     "JC_TRA_SLOW_FWD_LS";
      =     "JAMB_CLEANER_DB".TRA_SLOW_FWD_LS;
      A     L 0.0;
      A     "JC_TRA_SLOW_RET_LS";
      =     "JAMB_CLEANER_DB".TRA_SLOW_RET_LS;
      A     L 0.0;
      A     "TRA_NORMAL_FWD_LS";
      =     "JAMB_CLEANER_DB".TRA_NORM_FWD_LS;
      A     L 0.0;
      A     "TRA_NORMAL_RET_LS";
      =     "JAMB_CLEANER_DB".TRA_NORM_RET_LS;
      A     L 0.0;
      A     "VER_CLE_UP_LS";
      =     "JAMB_CLEANER_DB".VER_CLNR_UP_LS;
      A     L 0.0;
      A     "VER_CLE_DN_LS";
      =     "JAMB_CLEANER_DB".VER_CLNR_DN_LS;
      A     L 0.0;
      A(;
      A     "JAMB_CLNR_AUTO_STA_PB";
      A     "CTRL_SELECTION_CD";
      O;
      A     "WINCC_DB".CLN_OVN_JMB_AUTO_STA_PB;
      AN    "CTRL_SELECTION_CD";
      );
      =     "JAMB_CLEANER_DB".JAMB_CLNR_AUTO_STA_PB;
      A     L 0.0;
      A(;
      A     "JAMB_CLNR_AUTO_STP_PB";
      A     "CTRL_SELECTION_CD";
      O;
      A     "WINCC_DB".CLN_OVN_JMB_AUTO_STP_PB;
      AN    "CTRL_SELECTION_CD";
      );
      =     "JAMB_CLEANER_DB".JAMB_CLNR_AUTO_STP_PB;
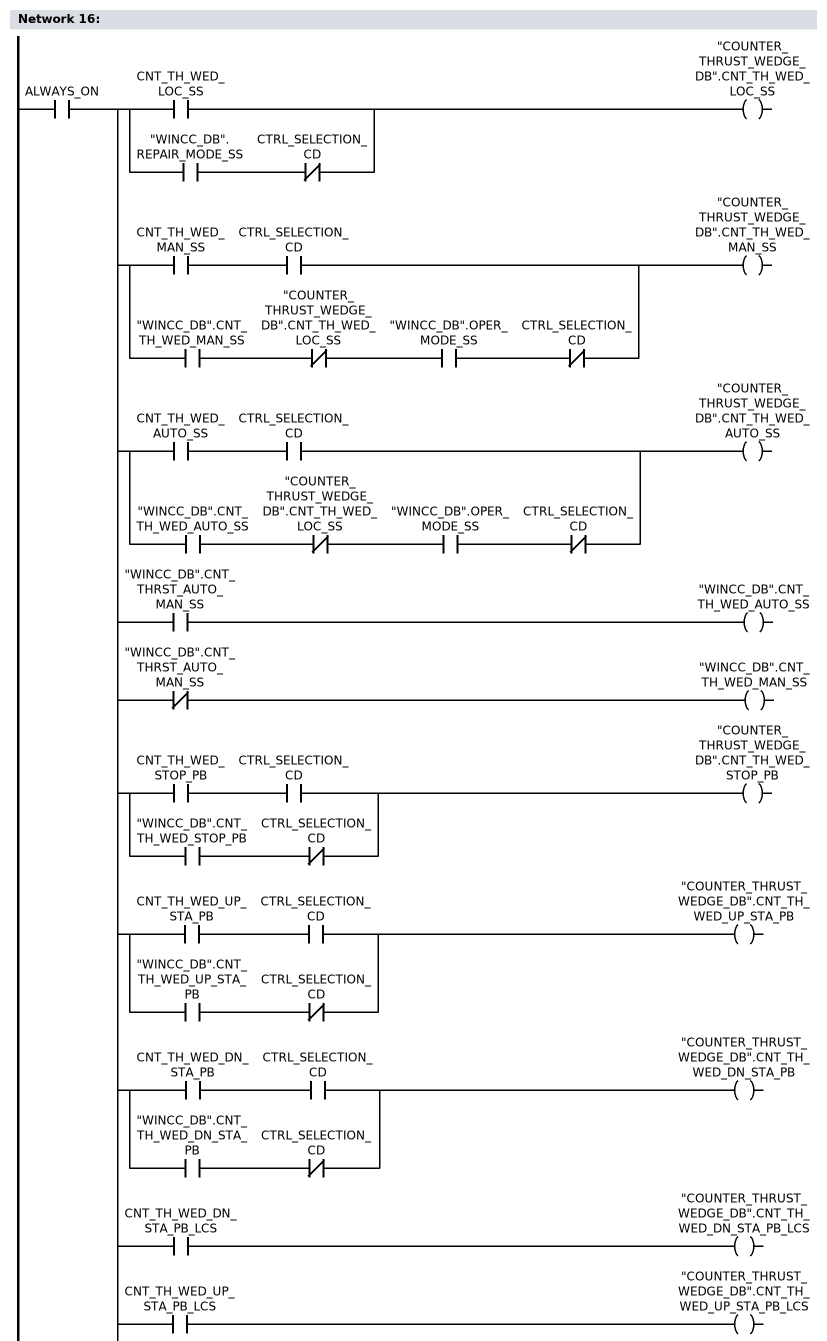
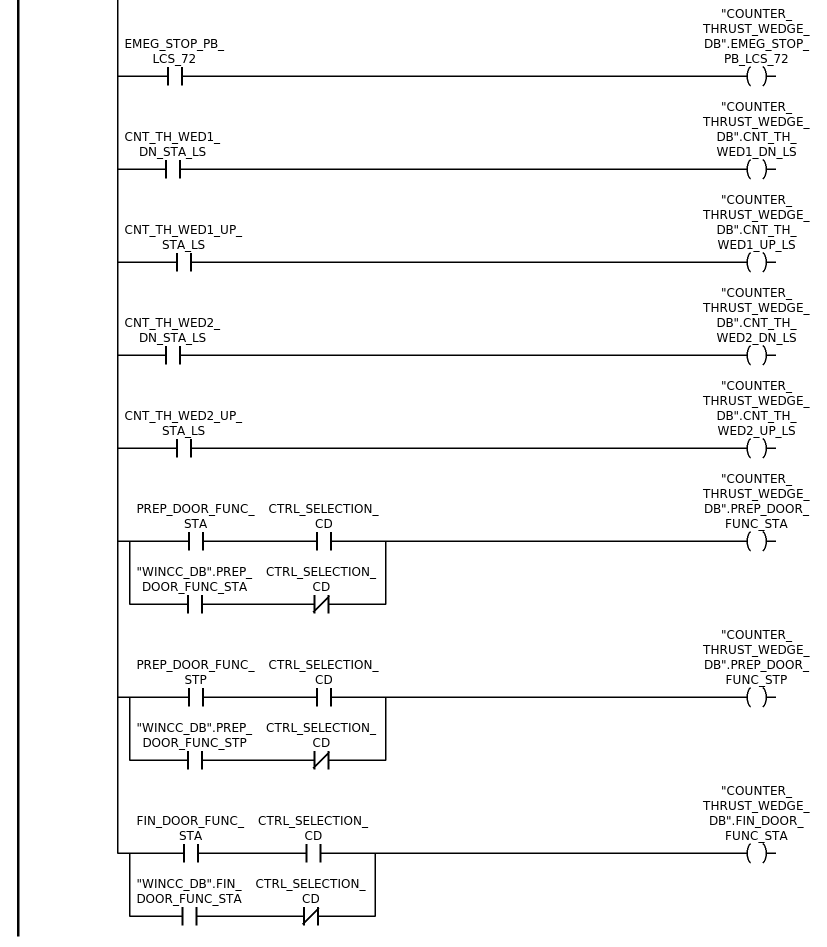
NETWORK
TITLE =
      A     "ALWAYS_ON";
      =     L 0.0;
      A     L 0.0;
      A(;
      O     "CNT_TH_WED_LOC_SS";
      O;
      A     "WINCC_DB".REPAIR_MODE_SS;
      AN    "CTRL_SELECTION_CD";
      );
      =     "COUNTER_THRUST_WEDGE_DB".CNT_TH_WED_LOC_SS;
      A     L 0.0;
      A(;
      A     "CNT_TH_WED_MAN_SS";
      A     "CTRL_SELECTION_CD";
      O;
      A     "WINCC_DB".CNT_TH_WED_MAN_SS;
      AN    "COUNTER_THRUST_WEDGE_DB".CNT_TH_WED_LOC_SS;
      A     "WINCC_DB".OPER_MODE_SS;
      AN    "CTRL_SELECTION_CD";
      );
      =     "COUNTER_THRUST_WEDGE_DB".CNT_TH_WED_MAN_SS;
      A     L 0.0;
      A(;
      A     "CNT_TH_WED_AUTO_SS";
      A     "CTRL_SELECTION_CD";
      O;
      A     "WINCC_DB".CNT_TH_WED_AUTO_SS;
      AN    "COUNTER_THRUST_WEDGE_DB".CNT_TH_WED_LOC_SS;
      A     "WINCC_DB".OPER_MODE_SS;
      AN    "CTRL_SELECTION_CD";
      );
      =     "COUNTER_THRUST_WEDGE_DB".CNT_TH_WED_AUTO_SS;
      A     L 0.0;
      A     "WINCC_DB".CNT_THRST_AUTO_MAN_SS;
      =     "WINCC_DB".CNT_TH_WED_AUTO_SS;
      A     L 0.0;
      AN    "WINCC_DB".CNT_THRST_AUTO_MAN_SS;
      =     "WINCC_DB".CNT_TH_WED_MAN_SS;
      A     L 0.0;
      A(;
      A     "CNT_TH_WED_STOP_PB";
      A     "CTRL_SELECTION_CD";
      O;
      A     "WINCC_DB".CNT_TH_WED_STOP_PB;
      AN    "CTRL_SELECTION_CD";
      );
      =     "COUNTER_THRUST_WEDGE_DB".CNT_TH_WED_STOP_PB;
      A     L 0.0;
      A(;
      A     "CNT_TH_WED_UP_STA_PB";
      A     "CTRL_SELECTION_CD";
      O;
      A     "WINCC_DB".CNT_TH_WED_UP_STA_PB;
      AN    "CTRL_SELECTION_CD";
      );
      =     "COUNTER_THRUST_WEDGE_DB".CNT_TH_WED_UP_STA_PB;
      A     L 0.0;
      A(;
      A     "CNT_TH_WED_DN_STA_PB";
      A     "CTRL_SELECTION_CD";
      O;
      A     "WINCC_DB".CNT_TH_WED_DN_STA_PB;
      AN    "CTRL_SELECTION_CD";
      );
      =     "COUNTER_THRUST_WEDGE_DB".CNT_TH_WED_DN_STA_PB;
      A     L 0.0;
      A     "CNT_TH_WED_DN_STA_PB_LCS";
      =     "COUNTER_THRUST_WEDGE_DB".CNT_TH_WED_DN_STA_PB_LCS;
      A     L 0.0;
      A     "CNT_TH_WED_UP_STA_PB_LCS";
      =     "COUNTER_THRUST_WEDGE_DB".CNT_TH_WED_UP_STA_PB_LCS;
      A     L 0.0;
      A     "EMEG_STOP_PB_LCS_72";
      =     "COUNTER_THRUST_WEDGE_DB".EMEG_STOP_PB_LCS_72;
      A     L 0.0;
      A     "CNT_TH_WED1_DN_STA_LS";
      =     "COUNTER_THRUST_WEDGE_DB".CNT_TH_WED1_DN_LS;
      A     L 0.0;
      A     "CNT_TH_WED1_UP_STA_LS";
      =     "COUNTER_THRUST_WEDGE_DB".CNT_TH_WED1_UP_LS;
      A     L 0.0;
      A     "CNT_TH_WED2_DN_STA_LS";
      =     "COUNTER_THRUST_WEDGE_DB".CNT_TH_WED2_DN_LS;
      A     L 0.0;
      A     "CNT_TH_WED2_UP_STA_LS";
      =     "COUNTER_THRUST_WEDGE_DB".CNT_TH_WED2_UP_LS;
      A     L 0.0;
      A(;
      A     "PREP_DOOR_FUNC_STA";
      A     "CTRL_SELECTION_CD";
      O;
      A     "WINCC_DB".PREP_DOOR_FUNC_STA;
      AN    "CTRL_SELECTION_CD";
      );
      =     "COUNTER_THRUST_WEDGE_DB".PREP_DOOR_FUNC_STA;
      A     L 0.0;
      A(;
      A     "PREP_DOOR_FUNC_STP";
      A     "CTRL_SELECTION_CD";
      O;
      A     "WINCC_DB".PREP_DOOR_FUNC_STP;
      AN    "CTRL_SELECTION_CD";
      );
      =     "COUNTER_THRUST_WEDGE_DB".PREP_DOOR_FUNC_STP;
      A     L 0.0;
      A(;
      A     "FIN_DOOR_FUNC_STA";
      A     "CTRL_SELECTION_CD";
      O;
      A     "WINCC_DB".FIN_DOOR_FUNC_STA;
      AN    "CTRL_SELECTION_CD";
      );
      =     "COUNTER_THRUST_WEDGE_DB".FIN_DOOR_FUNC_STA;
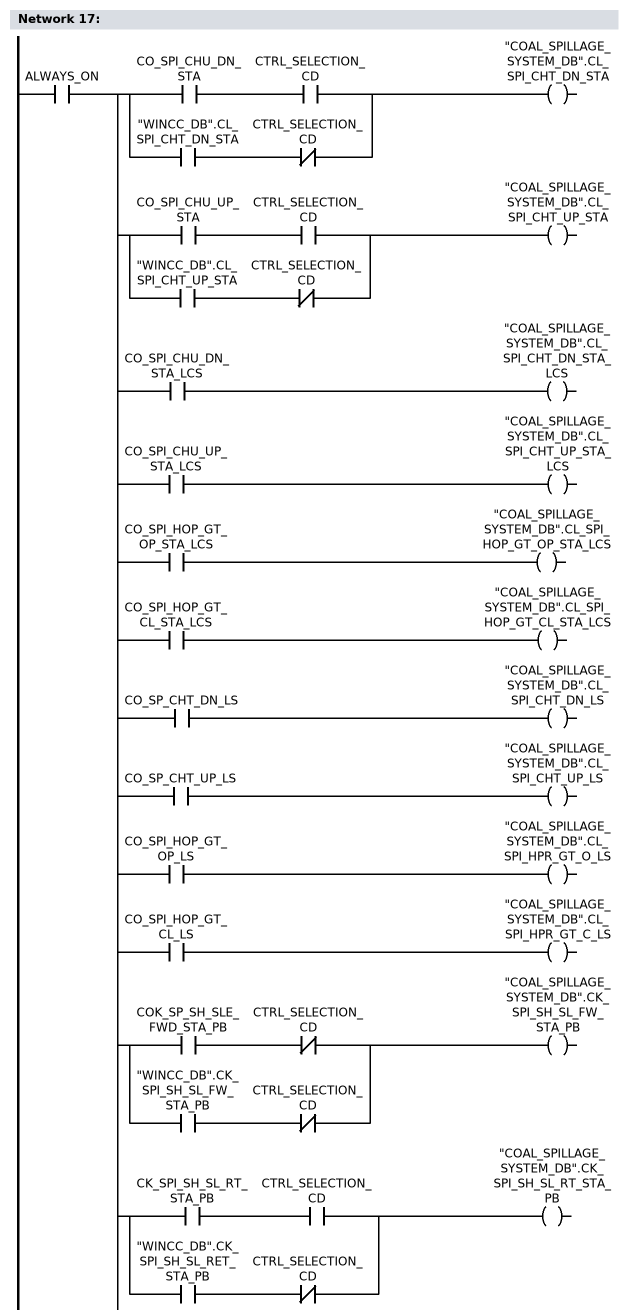
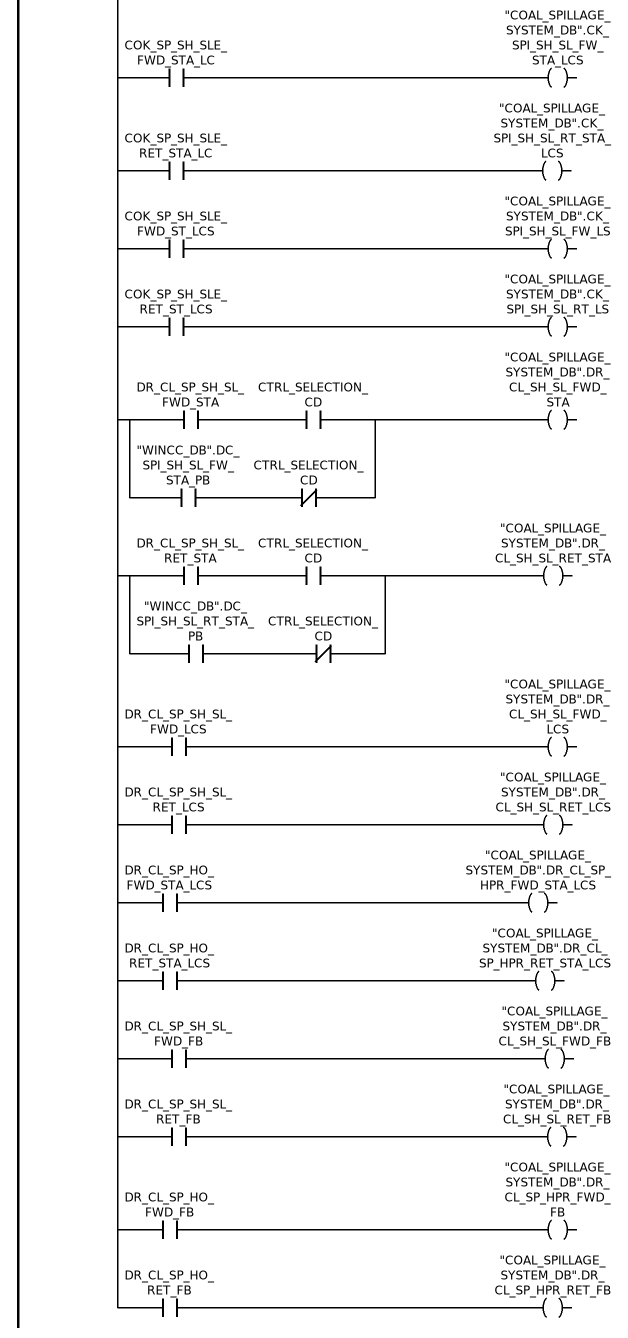
NETWORK
TITLE =
      A     "ALWAYS_ON";
      =     L 0.0;
      A     L 0.0;
      A(;
      A     "CO_SPI_CHU_DN_STA";
      A     "CTRL_SELECTION_CD";
      O;
      A     "WINCC_DB".CL_SPI_CHT_DN_STA;
      AN    "CTRL_SELECTION_CD";
      );
      =     "COAL_SPILLAGE_SYSTEM_DB".CL_SPI_CHT_DN_STA;
      A     L 0.0;
      A(;
      A     "CO_SPI_CHU_UP_STA";
      A     "CTRL_SELECTION_CD";
      O;
      A     "WINCC_DB".CL_SPI_CHT_UP_STA;
      AN    "CTRL_SELECTION_CD";
      );
      =     "COAL_SPILLAGE_SYSTEM_DB".CL_SPI_CHT_UP_STA;
      A     L 0.0;
      A     "CO_SPI_CHU_DN_STA_LCS";
      =     "COAL_SPILLAGE_SYSTEM_DB".CL_SPI_CHT_DN_STA_LCS;
      A     L 0.0;
      A     "CO_SPI_CHU_UP_STA_LCS";
      =     "COAL_SPILLAGE_SYSTEM_DB".CL_SPI_CHT_UP_STA_LCS;
      A     L 0.0;
      A     "CO_SPI_HOP_GT_OP_STA_LCS";
      =     "COAL_SPILLAGE_SYSTEM_DB".CL_SPI_HOP_GT_OP_STA_LCS;
      A     L 0.0;
      A     "CO_SPI_HOP_GT_CL_STA_LCS";
      =     "COAL_SPILLAGE_SYSTEM_DB".CL_SPI_HOP_GT_CL_STA_LCS;
      A     L 0.0;
      A     "CO_SP_CHT_DN_LS";
      =     "COAL_SPILLAGE_SYSTEM_DB".CL_SPI_CHT_DN_LS;
      A     L 0.0;
      A     "CO_SP_CHT_UP_LS";
      =     "COAL_SPILLAGE_SYSTEM_DB".CL_SPI_CHT_UP_LS;
      A     L 0.0;
      A     "CO_SPI_HOP_GT_OP_LS";
      =     "COAL_SPILLAGE_SYSTEM_DB".CL_SPI_HPR_GT_O_LS;
      A     L 0.0;
      A     "CO_SPI_HOP_GT_CL_LS";
      =     "COAL_SPILLAGE_SYSTEM_DB".CL_SPI_HPR_GT_C_LS;
      A     L 0.0;
      A(;
      A     "COK_SP_SH_SLE_FWD_STA_PB";
      AN    "CTRL_SELECTION_CD";
      O;
      A     "WINCC_DB".CK_SPI_SH_SL_FW_STA_PB;
      AN    "CTRL_SELECTION_CD";
      );
      =     "COAL_SPILLAGE_SYSTEM_DB".CK_SPI_SH_SL_FW_STA_PB;
      A     L 0.0;
      A(;
      A     "CK_SPI_SH_SL_RT_STA_PB";
      A     "CTRL_SELECTION_CD";
      O;
      A     "WINCC_DB".CK_SPI_SH_SL_RET_STA_PB;
      AN    "CTRL_SELECTION_CD";
      );
      =     "COAL_SPILLAGE_SYSTEM_DB".CK_SPI_SH_SL_RT_STA_PB;
      A     L 0.0;
      A     "COK_SP_SH_SLE_FWD_STA_LC";
      =     "COAL_SPILLAGE_SYSTEM_DB".CK_SPI_SH_SL_FW_STA_LCS;
      A     L 0.0;
      A     "COK_SP_SH_SLE_RET_STA_LC";
      =     "COAL_SPILLAGE_SYSTEM_DB".CK_SPI_SH_SL_RT_STA_LCS;
      A     L 0.0;
      A     "COK_SP_SH_SLE_FWD_ST_LCS";
      =     "COAL_SPILLAGE_SYSTEM_DB".CK_SPI_SH_SL_FW_LS;
      A     L 0.0;
      A     "COK_SP_SH_SLE_RET_ST_LCS";
      =     "COAL_SPILLAGE_SYSTEM_DB".CK_SPI_SH_SL_RT_LS;
      A     L 0.0;
      A(;
      A     "DR_CL_SP_SH_SL_FWD_STA";
      A     "CTRL_SELECTION_CD";
      O;
      A     "WINCC_DB".DC_SPI_SH_SL_FW_STA_PB;
      AN    "CTRL_SELECTION_CD";
      );
      =     "COAL_SPILLAGE_SYSTEM_DB".DR_CL_SH_SL_FWD_STA;
      A     L 0.0;
      A(;
      A     "DR_CL_SP_SH_SL_RET_STA";
      A     "CTRL_SELECTION_CD";
      O;
      A     "WINCC_DB".DC_SPI_SH_SL_RT_STA_PB;
      AN    "CTRL_SELECTION_CD";
      );
      =     "COAL_SPILLAGE_SYSTEM_DB".DR_CL_SH_SL_RET_STA;
      A     L 0.0;
      A     "DR_CL_SP_SH_SL_FWD_LCS";
      =     "COAL_SPILLAGE_SYSTEM_DB".DR_CL_SH_SL_FWD_LCS;
      A     L 0.0;
      A     "DR_CL_SP_SH_SL_RET_LCS";
      =     "COAL_SPILLAGE_SYSTEM_DB".DR_CL_SH_SL_RET_LCS;
      A     L 0.0;
      A     "DR_CL_SP_HO_FWD_STA_LCS";
      =     "COAL_SPILLAGE_SYSTEM_DB".DR_CL_SP_HPR_FWD_STA_LCS;
      A     L 0.0;
      A     "DR_CL_SP_HO_RET_STA_LCS";
      =     "COAL_SPILLAGE_SYSTEM_DB".DR_CL_SP_HPR_RET_STA_LCS;
      A     L 0.0;
      A     "DR_CL_SP_SH_SL_FWD_FB";
      =     "COAL_SPILLAGE_SYSTEM_DB".DR_CL_SH_SL_FWD_FB;
      A     L 0.0;
      A     "DR_CL_SP_SH_SL_RET_FB";
      =     "COAL_SPILLAGE_SYSTEM_DB".DR_CL_SH_SL_RET_FB;
      A     L 0.0;
      A     "DR_CL_SP_HO_FWD_FB";
      =     "COAL_SPILLAGE_SYSTEM_DB".DR_CL_SP_HPR_FWD_FB;
      A     L 0.0;
      A     "DR_CL_SP_HO_RET_FB";
      =     "COAL_SPILLAGE_SYSTEM_DB".DR_CL_SP_HPR_RET_FB;
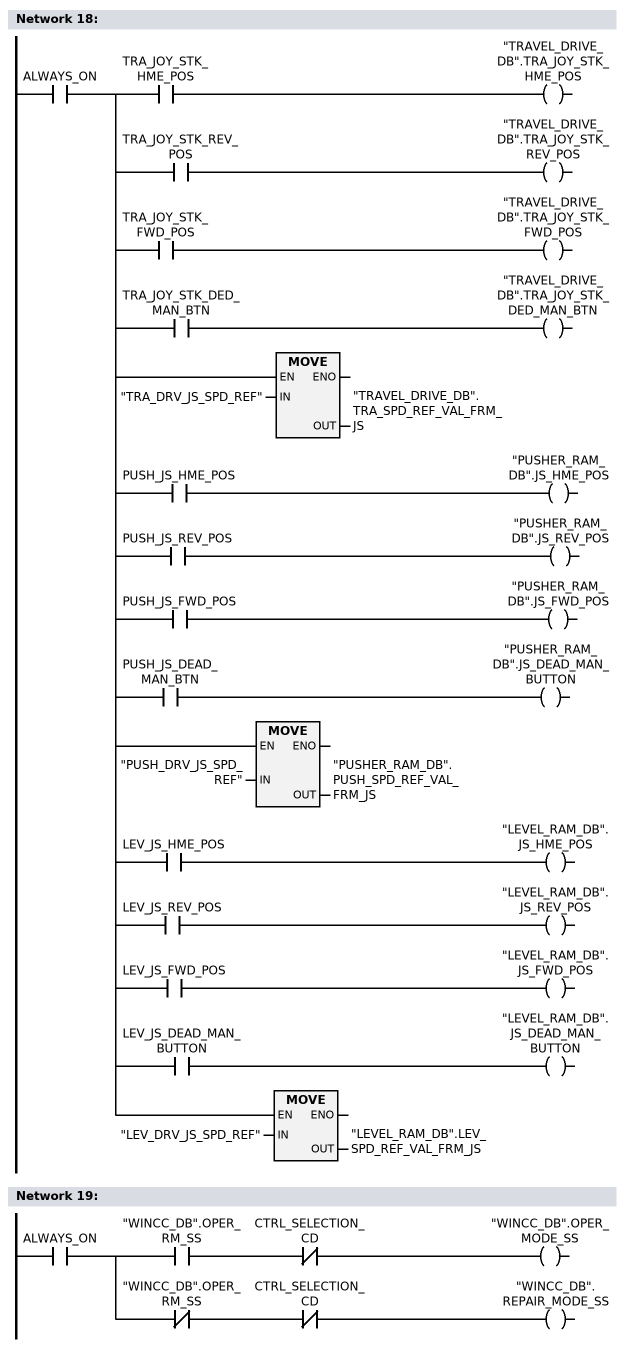
NETWORK
TITLE =
      A     "ALWAYS_ON";
      =     L 0.0;
      A     L 0.0;
      A     "TRA_JOY_STK_HME_POS";
      =     "TRAVEL_DRIVE_DB".TRA_JOY_STK_HME_POS;
      A     L 0.0;
      A     "TRA_JOY_STK_REV_POS";
      =     "TRAVEL_DRIVE_DB".TRA_JOY_STK_REV_POS;
      A     L 0.0;
      A     "TRA_JOY_STK_FWD_POS";
      =     "TRAVEL_DRIVE_DB".TRA_JOY_STK_FWD_POS;
      A     L 0.0;
      A     "TRA_JOY_STK_DED_MAN_BTN";
      =     "TRAVEL_DRIVE_DB".TRA_JOY_STK_DED_MAN_BTN;
      A     L 0.0;
      JNB   M001;
      L     "TRA_DRV_JS_SPD_REF";
      T     "TRAVEL_DRIVE_DB".TRA_SPD_REF_VAL_FRM_JS;
M001: NOP   0;
      A     L 0.0;
      A     "PUSH_JS_HME_POS";
      =     "PUSHER_RAM_DB".JS_HME_POS;
      A     L 0.0;
      A     "PUSH_JS_REV_POS";
      =     "PUSHER_RAM_DB".JS_REV_POS;
      A     L 0.0;
      A     "PUSH_JS_FWD_POS";
      =     "PUSHER_RAM_DB".JS_FWD_POS;
      A     L 0.0;
      A     "PUSH_JS_DEAD_MAN_BTN";
      =     "PUSHER_RAM_DB".JS_DEAD_MAN_BUTTON;
      A     L 0.0;
      JNB   M002;
      L     "PUSH_DRV_JS_SPD_REF";
      T     "PUSHER_RAM_DB".PUSH_SPD_REF_VAL_FRM_JS;
M002: NOP   0;
      A     L 0.0;
      A     "LEV_JS_HME_POS";
      =     "LEVEL_RAM_DB".JS_HME_POS;
      A     L 0.0;
      A     "LEV_JS_REV_POS";
      =     "LEVEL_RAM_DB".JS_REV_POS;
      A     L 0.0;
      A     "LEV_JS_FWD_POS";
      =     "LEVEL_RAM_DB".JS_FWD_POS;
      A     L 0.0;
      A     "LEV_JS_DEAD_MAN_BUTTON";
      =     "LEVEL_RAM_DB".JS_DEAD_MAN_BUTTON;
      A     L 0.0;
      JNB   M003;
      L     "LEV_DRV_JS_SPD_REF";
      T     "LEVEL_RAM_DB".LEV_SPD_REF_VAL_FRM_JS;
M003: NOP   0;
NETWORK
TITLE =
      A     "ALWAYS_ON";
      =     L 0.0;
      A     L 0.0;
      A     "WINCC_DB".OPER_RM_SS;
      AN    "CTRL_SELECTION_CD";
      =     "WINCC_DB".OPER_MODE_SS;
      A     L 0.0;
      AN    "WINCC_DB".OPER_RM_SS;
      AN    "CTRL_SELECTION_CD";
      =     "WINCC_DB".REPAIR_MODE_SS;
END_FUNCTION

FUNCTION "OUTPUT_MAPPING" : VOID	// FC 2
AUTHOR : Kamillas
VERSION : 0.1
BEGIN
// (block stored without names or comments; labels and parameter names are numbered)
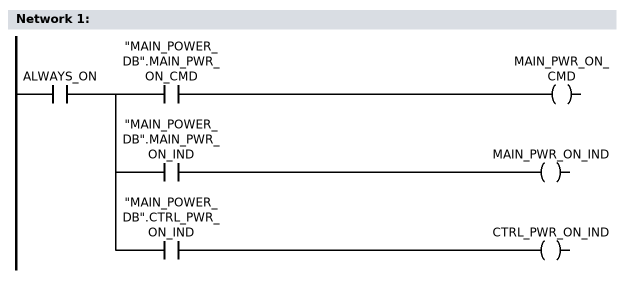
NETWORK
TITLE =
      A     "ALWAYS_ON";
      =     L 0.0;
      A     L 0.0;
      A     "MAIN_POWER_DB".MAIN_PWR_ON_CMD;
      =     "MAIN_PWR_ON_CMD";
      A     L 0.0;
      A     "MAIN_POWER_DB".MAIN_PWR_ON_IND;
      =     "MAIN_PWR_ON_IND";
      A     L 0.0;
      A     "MAIN_POWER_DB".CTRL_PWR_ON_IND;
      =     "CTRL_PWR_ON_IND";
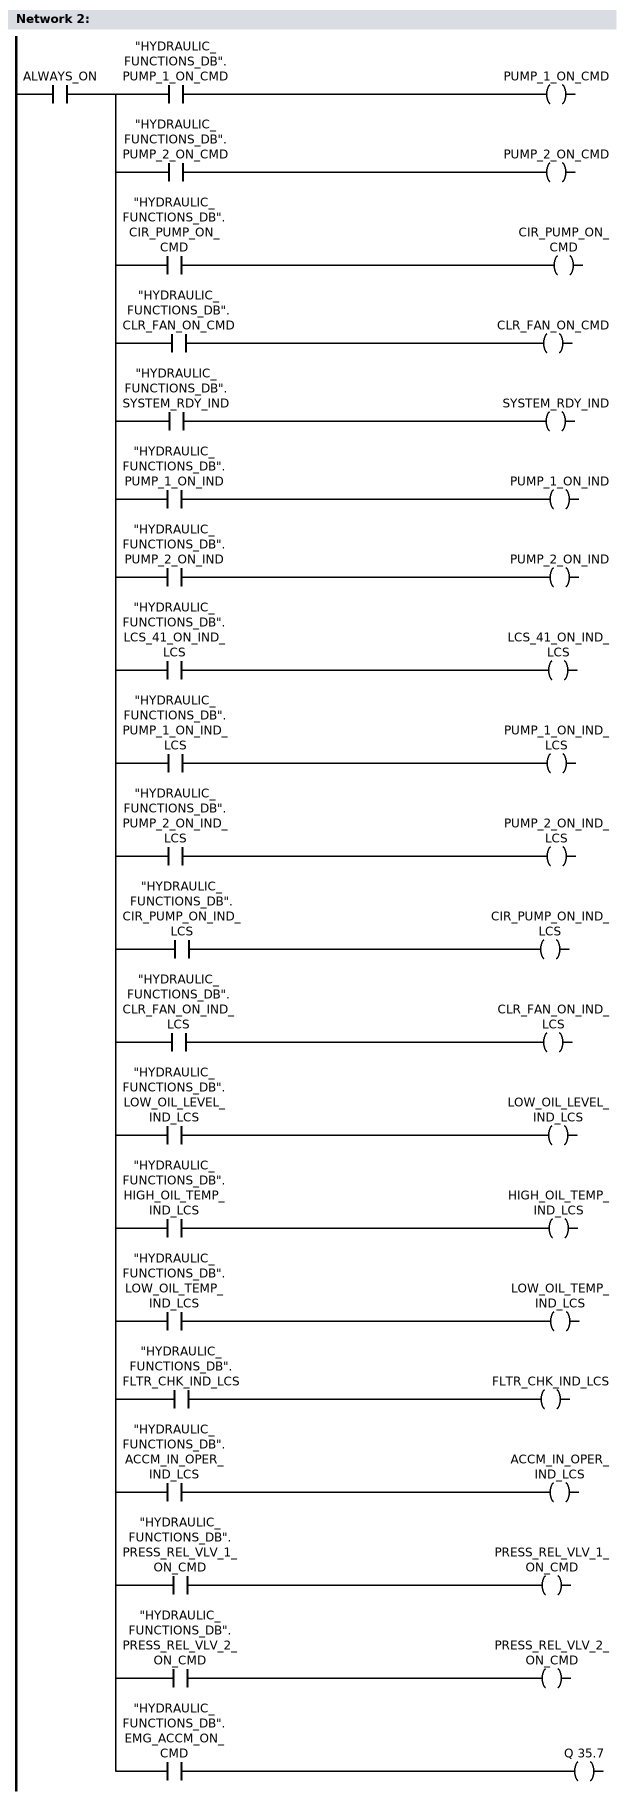
NETWORK
TITLE =
      A     "ALWAYS_ON";
      =     L 0.0;
      A     L 0.0;
      A     "HYDRAULIC_FUNCTIONS_DB".PUMP_1_ON_CMD;
      =     "PUMP_1_ON_CMD";
      A     L 0.0;
      A     "HYDRAULIC_FUNCTIONS_DB".PUMP_2_ON_CMD;
      =     "PUMP_2_ON_CMD";
      A     L 0.0;
      A     "HYDRAULIC_FUNCTIONS_DB".CIR_PUMP_ON_CMD;
      =     "CIR_PUMP_ON_CMD";
      A     L 0.0;
      A     "HYDRAULIC_FUNCTIONS_DB".CLR_FAN_ON_CMD;
      =     "CLR_FAN_ON_CMD";
      A     L 0.0;
      A     "HYDRAULIC_FUNCTIONS_DB".SYSTEM_RDY_IND;
      =     "SYSTEM_RDY_IND";
      A     L 0.0;
      A     "HYDRAULIC_FUNCTIONS_DB".PUMP_1_ON_IND;
      =     "PUMP_1_ON_IND";
      A     L 0.0;
      A     "HYDRAULIC_FUNCTIONS_DB".PUMP_2_ON_IND;
      =     "PUMP_2_ON_IND";
      A     L 0.0;
      A     "HYDRAULIC_FUNCTIONS_DB".LCS_41_ON_IND_LCS;
      =     "LCS_41_ON_IND_LCS";
      A     L 0.0;
      A     "HYDRAULIC_FUNCTIONS_DB".PUMP_1_ON_IND_LCS;
      =     "PUMP_1_ON_IND_LCS";
      A     L 0.0;
      A     "HYDRAULIC_FUNCTIONS_DB".PUMP_2_ON_IND_LCS;
      =     "PUMP_2_ON_IND_LCS";
      A     L 0.0;
      A     "HYDRAULIC_FUNCTIONS_DB".CIR_PUMP_ON_IND_LCS;
      =     "CIR_PUMP_ON_IND_LCS";
      A     L 0.0;
      A     "HYDRAULIC_FUNCTIONS_DB".CLR_FAN_ON_IND_LCS;
      =     "CLR_FAN_ON_IND_LCS";
      A     L 0.0;
      A     "HYDRAULIC_FUNCTIONS_DB".LOW_OIL_LEVEL_IND_LCS;
      =     "LOW_OIL_LEVEL_IND_LCS";
      A     L 0.0;
      A     "HYDRAULIC_FUNCTIONS_DB".HIGH_OIL_TEMP_IND_LCS;
      =     "HIGH_OIL_TEMP_IND_LCS";
      A     L 0.0;
      A     "HYDRAULIC_FUNCTIONS_DB".LOW_OIL_TEMP_IND_LCS;
      =     "LOW_OIL_TEMP_IND_LCS";
      A     L 0.0;
      A     "HYDRAULIC_FUNCTIONS_DB".FLTR_CHK_IND_LCS;
      =     "FLTR_CHK_IND_LCS";
      A     L 0.0;
      A     "HYDRAULIC_FUNCTIONS_DB".ACCM_IN_OPER_IND_LCS;
      =     "ACCM_IN_OPER_IND_LCS";
      A     L 0.0;
      A     "HYDRAULIC_FUNCTIONS_DB".PRESS_REL_VLV_1_ON_CMD;
      =     "PRESS_REL_VLV_1_ON_CMD";
      A     L 0.0;
      A     "HYDRAULIC_FUNCTIONS_DB".PRESS_REL_VLV_2_ON_CMD;
      =     "PRESS_REL_VLV_2_ON_CMD";
      A     L 0.0;
      A     "HYDRAULIC_FUNCTIONS_DB".EMG_ACCM_ON_CMD;
      =     Q 35.7;
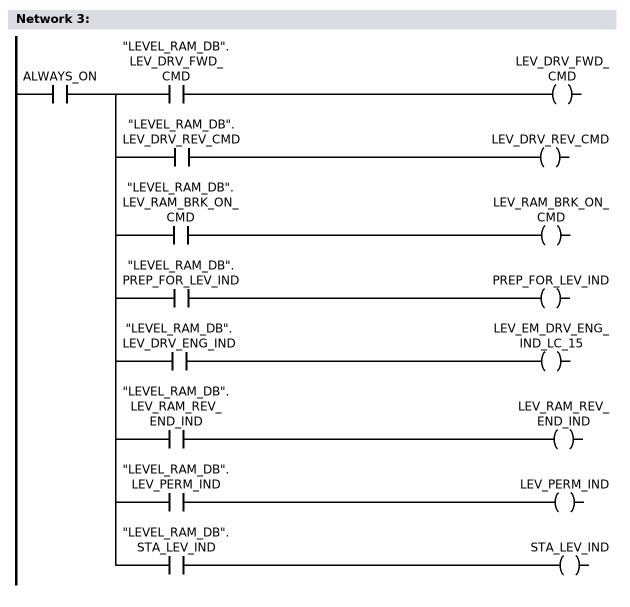
NETWORK
TITLE =
      A     "ALWAYS_ON";
      =     L 0.0;
      A     L 0.0;
      A     "LEVEL_RAM_DB".LEV_DRV_FWD_CMD;
      =     "LEV_DRV_FWD_CMD";
      A     L 0.0;
      A     "LEVEL_RAM_DB".LEV_DRV_REV_CMD;
      =     "LEV_DRV_REV_CMD";
      A     L 0.0;
      A     "LEVEL_RAM_DB".LEV_RAM_BRK_ON_CMD;
      =     "LEV_RAM_BRK_ON_CMD";
      A     L 0.0;
      A     "LEVEL_RAM_DB".PREP_FOR_LEV_IND;
      =     "PREP_FOR_LEV_IND";
      A     L 0.0;
      A     "LEVEL_RAM_DB".LEV_DRV_ENG_IND;
      =     "LEV_EM_DRV_ENG_IND_LC_15";
      A     L 0.0;
      A     "LEVEL_RAM_DB".LEV_RAM_REV_END_IND;
      =     "LEV_RAM_REV_END_IND";
      A     L 0.0;
      A     "LEVEL_RAM_DB".LEV_PERM_IND;
      =     "LEV_PERM_IND";
      A     L 0.0;
      A     "LEVEL_RAM_DB".STA_LEV_IND;
      =     "STA_LEV_IND";
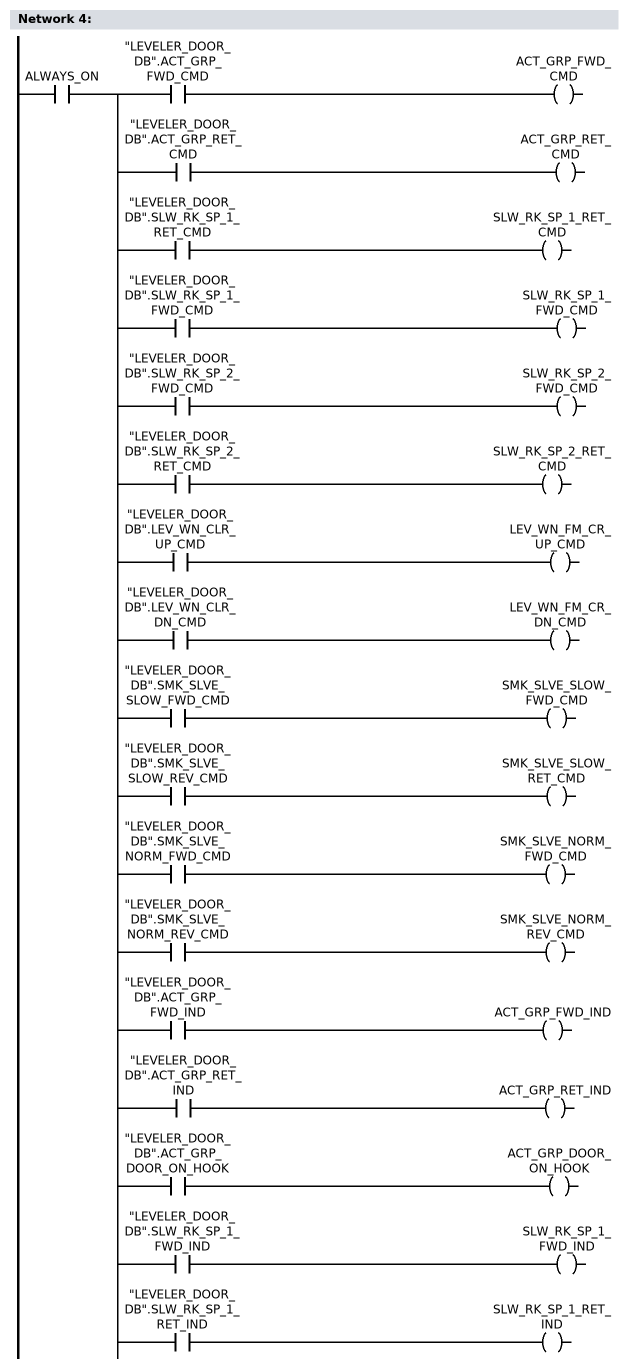
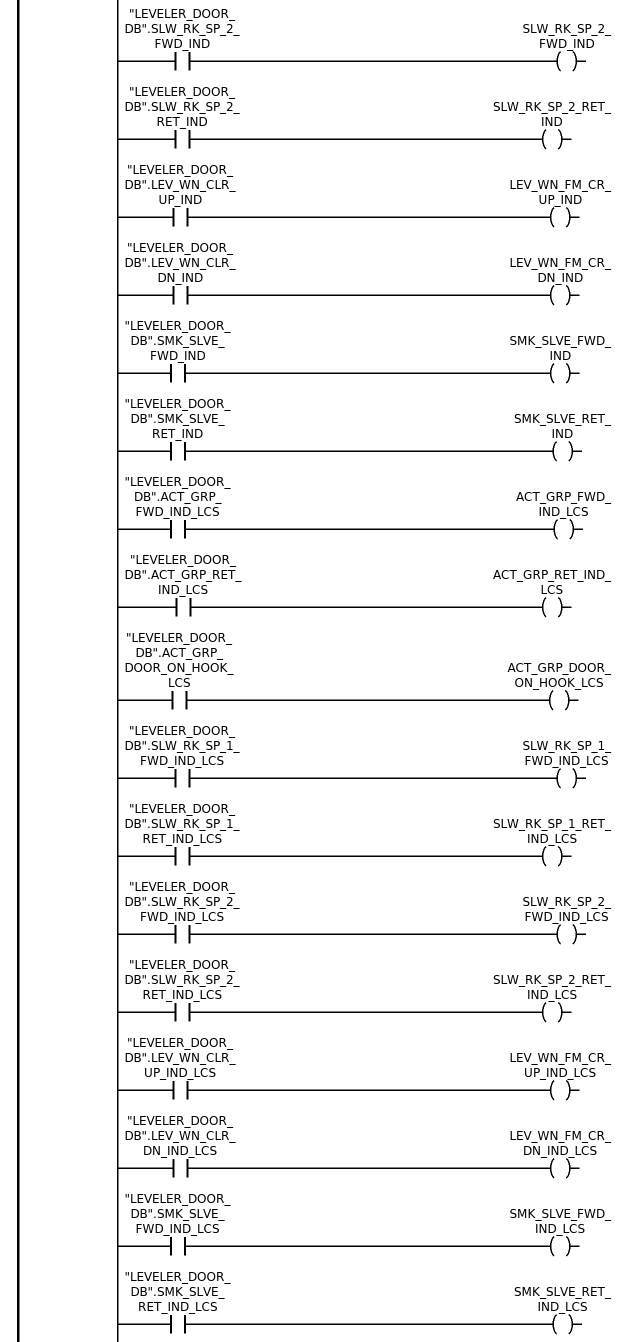
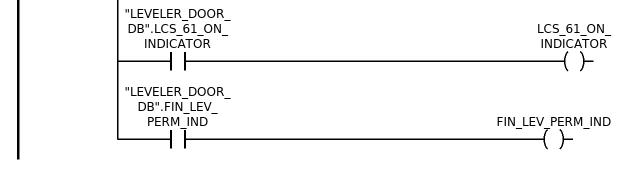
NETWORK
TITLE =
      A     "ALWAYS_ON";
      =     L 0.0;
      A     L 0.0;
      A     "LEVELER_DOOR_DB".ACT_GRP_FWD_CMD;
      =     "ACT_GRP_FWD_CMD";
      A     L 0.0;
      A     "LEVELER_DOOR_DB".ACT_GRP_RET_CMD;
      =     "ACT_GRP_RET_CMD";
      A     L 0.0;
      A     "LEVELER_DOOR_DB".SLW_RK_SP_1_RET_CMD;
      =     "SLW_RK_SP_1_RET_CMD";
      A     L 0.0;
      A     "LEVELER_DOOR_DB".SLW_RK_SP_1_FWD_CMD;
      =     "SLW_RK_SP_1_FWD_CMD";
      A     L 0.0;
      A     "LEVELER_DOOR_DB".SLW_RK_SP_2_FWD_CMD;
      =     "SLW_RK_SP_2_FWD_CMD";
      A     L 0.0;
      A     "LEVELER_DOOR_DB".SLW_RK_SP_2_RET_CMD;
      =     "SLW_RK_SP_2_RET_CMD";
      A     L 0.0;
      A     "LEVELER_DOOR_DB".LEV_WN_CLR_UP_CMD;
      =     "LEV_WN_FM_CR_UP_CMD";
      A     L 0.0;
      A     "LEVELER_DOOR_DB".LEV_WN_CLR_DN_CMD;
      =     "LEV_WN_FM_CR_DN_CMD";
      A     L 0.0;
      A     "LEVELER_DOOR_DB".SMK_SLVE_SLOW_FWD_CMD;
      =     "SMK_SLVE_SLOW_FWD_CMD";
      A     L 0.0;
      A     "LEVELER_DOOR_DB".SMK_SLVE_SLOW_REV_CMD;
      =     "SMK_SLVE_SLOW_RET_CMD";
      A     L 0.0;
      A     "LEVELER_DOOR_DB".SMK_SLVE_NORM_FWD_CMD;
      =     "SMK_SLVE_NORM_FWD_CMD";
      A     L 0.0;
      A     "LEVELER_DOOR_DB".SMK_SLVE_NORM_REV_CMD;
      =     "SMK_SLVE_NORM_REV_CMD";
      A     L 0.0;
      A     "LEVELER_DOOR_DB".ACT_GRP_FWD_IND;
      =     "ACT_GRP_FWD_IND";
      A     L 0.0;
      A     "LEVELER_DOOR_DB".ACT_GRP_RET_IND;
      =     "ACT_GRP_RET_IND";
      A     L 0.0;
      A     "LEVELER_DOOR_DB".ACT_GRP_DOOR_ON_HOOK;
      =     "ACT_GRP_DOOR_ON_HOOK";
      A     L 0.0;
      A     "LEVELER_DOOR_DB".SLW_RK_SP_1_FWD_IND;
      =     "SLW_RK_SP_1_FWD_IND";
      A     L 0.0;
      A     "LEVELER_DOOR_DB".SLW_RK_SP_1_RET_IND;
      =     "SLW_RK_SP_1_RET_IND";
      A     L 0.0;
      A     "LEVELER_DOOR_DB".SLW_RK_SP_2_FWD_IND;
      =     "SLW_RK_SP_2_FWD_IND";
      A     L 0.0;
      A     "LEVELER_DOOR_DB".SLW_RK_SP_2_RET_IND;
      =     "SLW_RK_SP_2_RET_IND";
      A     L 0.0;
      A     "LEVELER_DOOR_DB".LEV_WN_CLR_UP_IND;
      =     "LEV_WN_FM_CR_UP_IND";
      A     L 0.0;
      A     "LEVELER_DOOR_DB".LEV_WN_CLR_DN_IND;
      =     "LEV_WN_FM_CR_DN_IND";
      A     L 0.0;
      A     "LEVELER_DOOR_DB".SMK_SLVE_FWD_IND;
      =     "SMK_SLVE_FWD_IND";
      A     L 0.0;
      A     "LEVELER_DOOR_DB".SMK_SLVE_RET_IND;
      =     "SMK_SLVE_RET_IND";
      A     L 0.0;
      A     "LEVELER_DOOR_DB".ACT_GRP_FWD_IND_LCS;
      =     "ACT_GRP_FWD_IND_LCS";
      A     L 0.0;
      A     "LEVELER_DOOR_DB".ACT_GRP_RET_IND_LCS;
      =     "ACT_GRP_RET_IND_LCS";
      A     L 0.0;
      A     "LEVELER_DOOR_DB".ACT_GRP_DOOR_ON_HOOK_LCS;
      =     "ACT_GRP_DOOR_ON_HOOK_LCS";
      A     L 0.0;
      A     "LEVELER_DOOR_DB".SLW_RK_SP_1_FWD_IND_LCS;
      =     "SLW_RK_SP_1_FWD_IND_LCS";
      A     L 0.0;
      A     "LEVELER_DOOR_DB".SLW_RK_SP_1_RET_IND_LCS;
      =     "SLW_RK_SP_1_RET_IND_LCS";
      A     L 0.0;
      A     "LEVELER_DOOR_DB".SLW_RK_SP_2_FWD_IND_LCS;
      =     "SLW_RK_SP_2_FWD_IND_LCS";
      A     L 0.0;
      A     "LEVELER_DOOR_DB".SLW_RK_SP_2_RET_IND_LCS;
      =     "SLW_RK_SP_2_RET_IND_LCS";
      A     L 0.0;
      A     "LEVELER_DOOR_DB".LEV_WN_CLR_UP_IND_LCS;
      =     "LEV_WN_FM_CR_UP_IND_LCS";
      A     L 0.0;
      A     "LEVELER_DOOR_DB".LEV_WN_CLR_DN_IND_LCS;
      =     "LEV_WN_FM_CR_DN_IND_LCS";
      A     L 0.0;
      A     "LEVELER_DOOR_DB".SMK_SLVE_FWD_IND_LCS;
      =     "SMK_SLVE_FWD_IND_LCS";
      A     L 0.0;
      A     "LEVELER_DOOR_DB".SMK_SLVE_RET_IND_LCS;
      =     "SMK_SLVE_RET_IND_LCS";
      A     L 0.0;
      A     "LEVELER_DOOR_DB".LCS_61_ON_INDICATOR;
      =     "LCS_61_ON_INDICATOR";
      A     L 0.0;
      A     "LEVELER_DOOR_DB".FIN_LEV_PERM_IND;
      =     "FIN_LEV_PERM_IND";
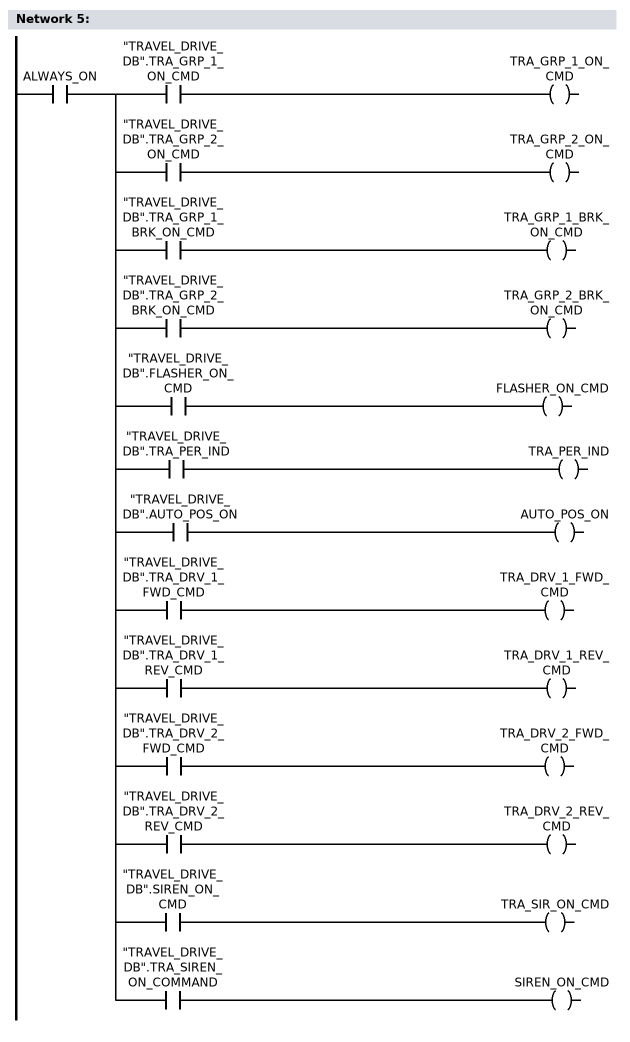
NETWORK
TITLE =
      A     "ALWAYS_ON";
      =     L 0.0;
      A     L 0.0;
      A     "TRAVEL_DRIVE_DB".TRA_GRP_1_ON_CMD;
      =     "TRA_GRP_1_ON_CMD";
      A     L 0.0;
      A     "TRAVEL_DRIVE_DB".TRA_GRP_2_ON_CMD;
      =     "TRA_GRP_2_ON_CMD";
      A     L 0.0;
      A     "TRAVEL_DRIVE_DB".TRA_GRP_1_BRK_ON_CMD;
      =     "TRA_GRP_1_BRK_ON_CMD";
      A     L 0.0;
      A     "TRAVEL_DRIVE_DB".TRA_GRP_2_BRK_ON_CMD;
      =     "TRA_GRP_2_BRK_ON_CMD";
      A     L 0.0;
      A     "TRAVEL_DRIVE_DB".FLASHER_ON_CMD;
      =     "FLASHER_ON_CMD";
      A     L 0.0;
      A     "TRAVEL_DRIVE_DB".TRA_PER_IND;
      =     "TRA_PER_IND";
      A     L 0.0;
      A     "TRAVEL_DRIVE_DB".AUTO_POS_ON;
      =     "AUTO_POS_ON";
      A     L 0.0;
      A     "TRAVEL_DRIVE_DB".TRA_DRV_1_FWD_CMD;
      =     "TRA_DRV_1_FWD_CMD";
      A     L 0.0;
      A     "TRAVEL_DRIVE_DB".TRA_DRV_1_REV_CMD;
      =     "TRA_DRV_1_REV_CMD";
      A     L 0.0;
      A     "TRAVEL_DRIVE_DB".TRA_DRV_2_FWD_CMD;
      =     "TRA_DRV_2_FWD_CMD";
      A     L 0.0;
      A     "TRAVEL_DRIVE_DB".TRA_DRV_2_REV_CMD;
      =     "TRA_DRV_2_REV_CMD";
      A     L 0.0;
      A     "TRAVEL_DRIVE_DB".SIREN_ON_CMD;
      =     "TRA_SIR_ON_CMD";
      A     L 0.0;
      A     "TRAVEL_DRIVE_DB".TRA_SIREN_ON_COMMAND;
      =     "SIREN_ON_CMD";
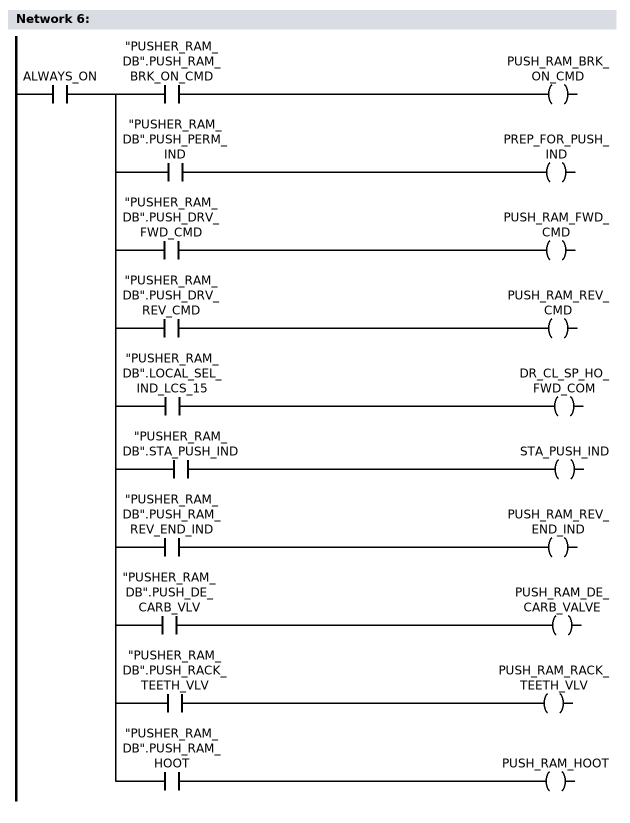
NETWORK
TITLE =
      A     "ALWAYS_ON";
      =     L 0.0;
      A     L 0.0;
      A     "PUSHER_RAM_DB".PUSH_RAM_BRK_ON_CMD;
      =     "PUSH_RAM_BRK_ON_CMD";
      A     L 0.0;
      A     "PUSHER_RAM_DB".PUSH_PERM_IND;
      =     "PREP_FOR_PUSH_IND";
      A     L 0.0;
      A     "PUSHER_RAM_DB".PUSH_DRV_FWD_CMD;
      =     "PUSH_RAM_FWD_CMD";
      A     L 0.0;
      A     "PUSHER_RAM_DB".PUSH_DRV_REV_CMD;
      =     "PUSH_RAM_REV_CMD";
      A     L 0.0;
      A     "PUSHER_RAM_DB".LOCAL_SEL_IND_LCS_15;
      =     "DR_CL_SP_HO_FWD_COM";
      A     L 0.0;
      A     "PUSHER_RAM_DB".STA_PUSH_IND;
      =     "STA_PUSH_IND";
      A     L 0.0;
      A     "PUSHER_RAM_DB".PUSH_RAM_REV_END_IND;
      =     "PUSH_RAM_REV_END_IND";
      A     L 0.0;
      A     "PUSHER_RAM_DB".PUSH_DE_CARB_VLV;
      =     "PUSH_RAM_DE_CARB_VALVE";
      A     L 0.0;
      A     "PUSHER_RAM_DB".PUSH_RACK_TEETH_VLV;
      =     "PUSH_RAM_RACK_TEETH_VLV";
      A     L 0.0;
      A     "PUSHER_RAM_DB".PUSH_RAM_HOOT;
      =     "PUSH_RAM_HOOT";
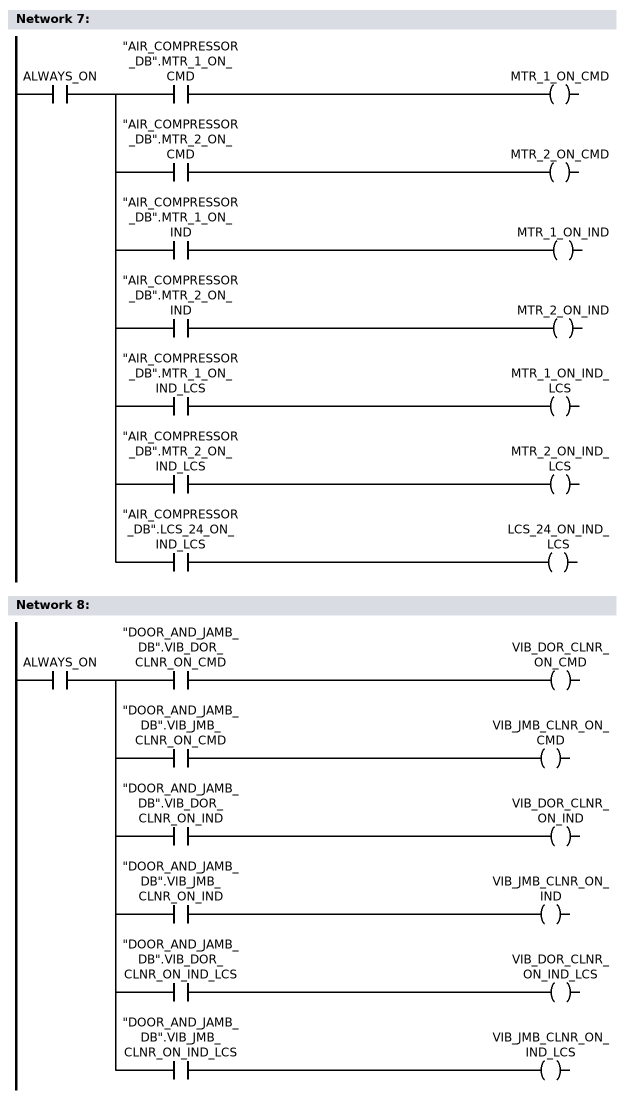
NETWORK
TITLE =
      A     "ALWAYS_ON";
      =     L 0.0;
      A     L 0.0;
      A     "AIR_COMPRESSOR_DB".MTR_1_ON_CMD;
      =     "MTR_1_ON_CMD";
      A     L 0.0;
      A     "AIR_COMPRESSOR_DB".MTR_2_ON_CMD;
      =     "MTR_2_ON_CMD";
      A     L 0.0;
      A     "AIR_COMPRESSOR_DB".MTR_1_ON_IND;
      =     "MTR_1_ON_IND";
      A     L 0.0;
      A     "AIR_COMPRESSOR_DB".MTR_2_ON_IND;
      =     "MTR_2_ON_IND";
      A     L 0.0;
      A     "AIR_COMPRESSOR_DB".MTR_1_ON_IND_LCS;
      =     "MTR_1_ON_IND_LCS";
      A     L 0.0;
      A     "AIR_COMPRESSOR_DB".MTR_2_ON_IND_LCS;
      =     "MTR_2_ON_IND_LCS";
      A     L 0.0;
      A     "AIR_COMPRESSOR_DB".LCS_24_ON_IND_LCS;
      =     "LCS_24_ON_IND_LCS";
NETWORK
TITLE =
      A     "ALWAYS_ON";
      =     L 0.0;
      A     L 0.0;
      A     "DOOR_AND_JAMB_DB".VIB_DOR_CLNR_ON_CMD;
      =     "VIB_DOR_CLNR_ON_CMD";
      A     L 0.0;
      A     "DOOR_AND_JAMB_DB".VIB_JMB_CLNR_ON_CMD;
      =     "VIB_JMB_CLNR_ON_CMD";
      A     L 0.0;
      A     "DOOR_AND_JAMB_DB".VIB_DOR_CLNR_ON_IND;
      =     "VIB_DOR_CLNR_ON_IND";
      A     L 0.0;
      A     "DOOR_AND_JAMB_DB".VIB_JMB_CLNR_ON_IND;
      =     "VIB_JMB_CLNR_ON_IND";
      A     L 0.0;
      A     "DOOR_AND_JAMB_DB".VIB_DOR_CLNR_ON_IND_LCS;
      =     "VIB_DOR_CLNR_ON_IND_LCS";
      A     L 0.0;
      A     "DOOR_AND_JAMB_DB".VIB_JMB_CLNR_ON_IND_LCS;
      =     "VIB_JMB_CLNR_ON_IND_LCS";
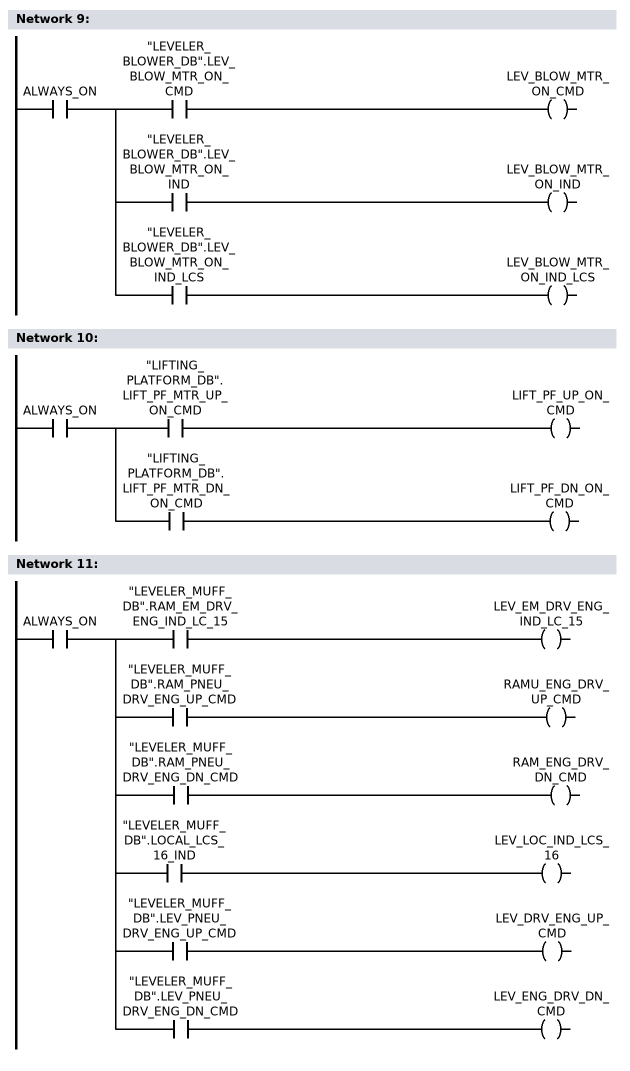
NETWORK
TITLE =
      A     "ALWAYS_ON";
      =     L 0.0;
      A     L 0.0;
      A     "LEVELER_BLOWER_DB".LEV_BLOW_MTR_ON_CMD;
      =     "LEV_BLOW_MTR_ON_CMD";
      A     L 0.0;
      A     "LEVELER_BLOWER_DB".LEV_BLOW_MTR_ON_IND;
      =     "LEV_BLOW_MTR_ON_IND";
      A     L 0.0;
      A     "LEVELER_BLOWER_DB".LEV_BLOW_MTR_ON_IND_LCS;
      =     "LEV_BLOW_MTR_ON_IND_LCS";
NETWORK
TITLE =
      A     "ALWAYS_ON";
      =     L 0.0;
      A     L 0.0;
      A     "LIFTING_PLATFORM_DB".LIFT_PF_MTR_UP_ON_CMD;
      =     "LIFT_PF_UP_ON_CMD";
      A     L 0.0;
      A     "LIFTING_PLATFORM_DB".LIFT_PF_MTR_DN_ON_CMD;
      =     "LIFT_PF_DN_ON_CMD";
NETWORK
TITLE =
      A     "ALWAYS_ON";
      =     L 0.0;
      A     L 0.0;
      A     "LEVELER_MUFF_DB".RAM_EM_DRV_ENG_IND_LC_15;
      =     "LEV_EM_DRV_ENG_IND_LC_15";
      A     L 0.0;
      A     "LEVELER_MUFF_DB".RAM_PNEU_DRV_ENG_UP_CMD;
      =     "RAMU_ENG_DRV_UP_CMD";
      A     L 0.0;
      A     "LEVELER_MUFF_DB".RAM_PNEU_DRV_ENG_DN_CMD;
      =     "RAM_ENG_DRV_DN_CMD";
      A     L 0.0;
      A     "LEVELER_MUFF_DB".LOCAL_LCS_16_IND;
      =     "LEV_LOC_IND_LCS_16";
      A     L 0.0;
      A     "LEVELER_MUFF_DB".LEV_PNEU_DRV_ENG_UP_CMD;
      =     "LEV_DRV_ENG_UP_CMD";
      A     L 0.0;
      A     "LEVELER_MUFF_DB".LEV_PNEU_DRV_ENG_DN_CMD;
      =     "LEV_ENG_DRV_DN_CMD";
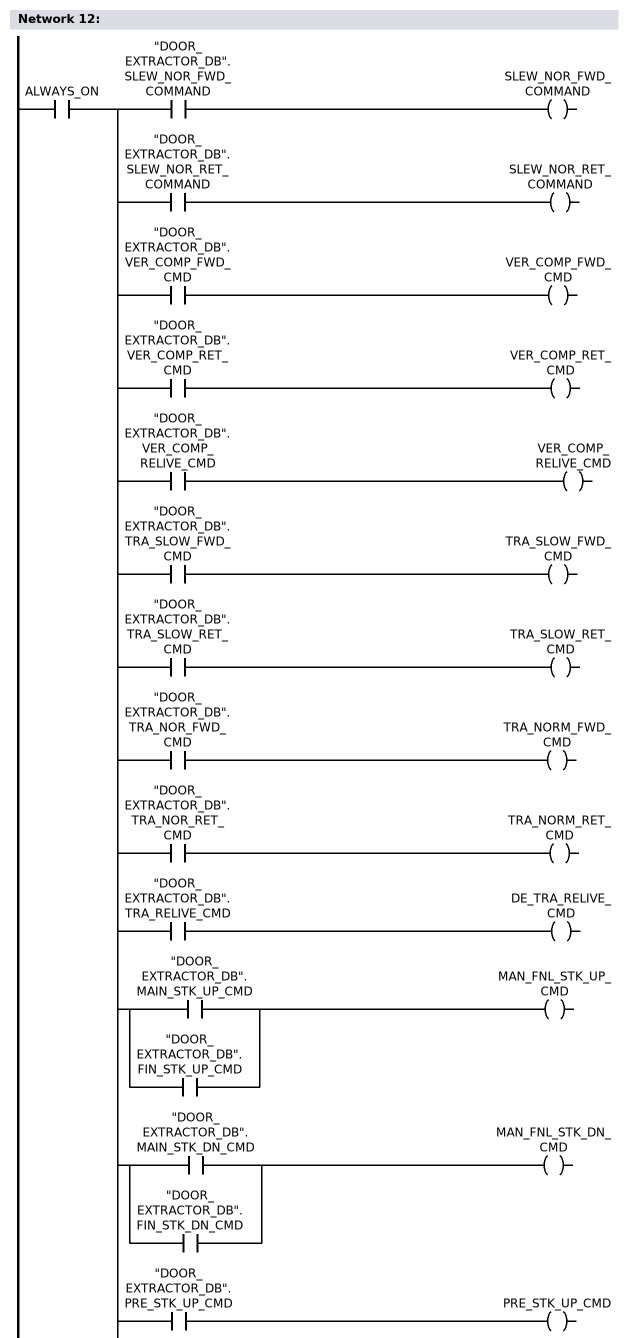
